{region " SIGNAL AREA : NAME->X_I_Out_ESS LENGTH->16 STARTBIT :48"}
_FB_UNPACK_WORD_TO_BYTE_6 (
		X_WORD_0										:= 
(*SELECT 1 : Is data valid and range is not exceed?*)	SEL((GVL.IOVD.X_I_Out_ESS.v AND NOT GVL.IOVD.X_I_Out_ESS.RangeExcd),
(*SELECT 2 : Is NOT AVAILABLE ?*)						SEL(GVL.IOVD.X_I_Out_ESS.na,
(*SELECT 3 : Is ERROR active ?*)						SEL(GVL.IOVD.X_I_Out_ESS.e,
(*DEFAULT VALUE assignment*)							UINT_TO_WORD(REAL_TO_UINT((32766))),
(*ERROR is active*)										16#FEFE),
(*NOT AVAILABLE is active*)								16#FFFF),
(*Transmission is VALID*)								UINT_TO_WORD(REAL_TO_UINT((GVL.IOVD.X_I_Out_ESS.x + 32766)))),
		X_BYTE_0										=> _FB_CanTx_Message_463.X_Byte_6,
		X_BYTE_1										=> _FB_CanTx_Message_463.X_Byte_7);
{endregion}

_FB_CanTx_Message_463.X_Byte_3 		:= 16#FF;

_FB_CanTx_Message_463 (		C_Enable		:= GVL.IOVD.C_En_TCU_Analog_0X463,
     						Obj_CAN			:= ADR(GVL.IC.Obj_CAN0),
     						X_MsgID			:= 16#463,
     						Tm_CycleTime	:= TIME#250MS,
     						N_Msg_Dlc		:= 8,
     						S_Extended		:= 0,
     						S_Sent_Ok   	=> GVL.IOVD.S_SentOk_TCU_Analog_0X463);
{endregion}
//-----------------------------------------------------------------------------------------------------------------------------
//-----------------------------------------------------------------------------------------------------------------------------
{region " MESSAGE AREA :TCU_Cikis_Akim_Guc- ID:464"}

{region " SIGNAL AREA : NAME->X_I_Out_Mot_Cnv LENGTH->16 STARTBIT :0"}
_FB_UNPACK_WORD_TO_BYTE_7(
		X_WORD_0										:= 
(*SELECT 1 : Is data valid and range is not exceed?*)	SEL((GVL.IOVD.X_I_Out_Mot_Cnv.v AND NOT GVL.IOVD.X_I_Out_Mot_Cnv.RangeExcd),
(*SELECT 2 : Is NOT AVAILABLE ?*)						SEL(GVL.IOVD.X_I_Out_Mot_Cnv.na,
(*SELECT 3 : Is ERROR active ?*)						SEL(GVL.IOVD.X_I_Out_Mot_Cnv.e,
(*DEFAULT VALUE assignment*)							UINT_TO_WORD(REAL_TO_UINT((1600)/0.05)),
(*ERROR is active*)										16#FEFE),
(*NOT AVAILABLE is active*)								16#FFFF),
(*Transmission is VALID*)								UINT_TO_WORD(REAL_TO_UINT((GVL.IOVD.X_I_Out_Mot_Cnv.x + 1600)/0.05))),
		X_BYTE_0										=> _FB_CanTx_Message_464.X_Byte_0,
		X_BYTE_1										=> _FB_CanTx_Message_464.X_Byte_1);
{endregion}

{region " SIGNAL AREA : NAME->X_I_Brk_Rsr LENGTH->16 STARTBIT :16"}
_FB_UNPACK_WORD_TO_BYTE_8(
		X_WORD_0										:= 
(*SELECT 1 : Is data valid and range is not exceed?*)	SEL((GVL.IOVD.X_I_Brk_Rsr.v AND NOT GVL.IOVD.X_I_Brk_Rsr.RangeExcd),
(*SELECT 2 : Is NOT AVAILABLE ?*)						SEL(GVL.IOVD.X_I_Brk_Rsr.na,
(*SELECT 3 : Is ERROR active ?*)						SEL(GVL.IOVD.X_I_Brk_Rsr.e,
(*DEFAULT VALUE assignment*)							UINT_TO_WORD(REAL_TO_UINT((1600)/0.05)),
(*ERROR is active*)										16#FEFE),
(*NOT AVAILABLE is active*)								16#FFFF),
(*Transmission is VALID*)								UINT_TO_WORD(REAL_TO_UINT((GVL.IOVD.X_I_Brk_Rsr.x + 1600)/0.05))),
		X_BYTE_0										=> _FB_CanTx_Message_464.X_Byte_2,
		X_BYTE_1										=> _FB_CanTx_Message_464.X_Byte_3);
{endregion}

{region " SIGNAL AREA : NAME->X_P_Mot_Cnv LENGTH->16 STARTBIT :32"}
_FB_UNPACK_WORD_TO_BYTE_9(
		X_WORD_0										:= 
(*SELECT 1 : Is data valid and range is not exceed?*)	SEL((GVL.IOVD.X_P_Mot_Cnv.v AND NOT GVL.IOVD.X_P_Mot_Cnv.RangeExcd),
(*SELECT 2 : Is NOT AVAILABLE ?*)						SEL(GVL.IOVD.X_P_Mot_Cnv.na,
(*SELECT 3 : Is ERROR active ?*)						SEL(GVL.IOVD.X_P_Mot_Cnv.e,
(*DEFAULT VALUE assignment*)							UINT_TO_WORD(REAL_TO_UINT((750)/0.025)),
(*ERROR is active*)										16#FEFE),
(*NOT AVAILABLE is active*)								16#FFFF),
(*Transmission is VALID*)								UINT_TO_WORD(REAL_TO_UINT((GVL.IOVD.X_P_Mot_Cnv.x + 750)/0.025))),
		X_BYTE_0										=> _FB_CanTx_Message_464.X_Byte_4,
		X_BYTE_1										=> _FB_CanTx_Message_464.X_Byte_5);
{endregion}

{region " SIGNAL AREA : NAME->X_P_Brk_Rsr LENGTH->16 STARTBIT :48"}
_FB_UNPACK_WORD_TO_BYTE_10(
		X_WORD_0										:= 
(*SELECT 1 : Is data valid and range is not exceed?*)	SEL((GVL.IOVD.X_P_Brk_Rsr.v AND NOT GVL.IOVD.X_P_Brk_Rsr.RangeExcd),
(*SELECT 2 : Is NOT AVAILABLE ?*)						SEL(GVL.IOVD.X_P_Brk_Rsr.na,
(*SELECT 3 : Is ERROR active ?*)						SEL(GVL.IOVD.X_P_Brk_Rsr.e,
(*DEFAULT VALUE assignment*)							UINT_TO_WORD(REAL_TO_UINT((750)/0.025)),
(*ERROR is active*)										16#FEFE),
(*NOT AVAILABLE is active*)								16#FFFF),
(*Transmission is VALID*)								UINT_TO_WORD(REAL_TO_UINT((GVL.IOVD.X_P_Brk_Rsr.x + 750)/0.025))),
		X_BYTE_0										=> _FB_CanTx_Message_464.X_Byte_6,
		X_BYTE_1										=> _FB_CanTx_Message_464.X_Byte_7);
{endregion}

_FB_CanTx_Message_464 (		C_Enable		:= GVL.IOVD.C_En_TCU_Cikis_Akim_Guc_0X464,
     						Obj_CAN			:= ADR(GVL.IC.Obj_CAN0),
     						X_MsgID			:= 16#464,
     						Tm_CycleTime	:= TIME#250MS,
     						N_Msg_Dlc		:= 8,
     						S_Extended		:= 0,
     						S_Sent_Ok   	=> GVL.IOVD.S_SentOk_TCU_Cikis_Akim_Guc_0X464);
{endregion}
//-----------------------------------------------------------------------------------------------------------------------------
//-----------------------------------------------------------------------------------------------------------------------------
{region " MESSAGE AREA :TCU_Tork_Hiz- ID:465"}

{region " SIGNAL AREA : NAME->X_M_Act LENGTH->16 STARTBIT :0"}
_FB_UNPACK_WORD_TO_BYTE_11 (
		X_WORD_0										:= 
(*SELECT 1 : Is data valid and range is not exceed?*)	SEL((GVL.IOVD.X_M_Act.v AND NOT GVL.IOVD.X_M_Act.RangeExcd),
(*SELECT 2 : Is NOT AVAILABLE ?*)						SEL(GVL.IOVD.X_M_Act.na,
(*SELECT 3 : Is ERROR active ?*)						SEL(GVL.IOVD.X_M_Act.e,
(*DEFAULT VALUE assignment*)							UINT_TO_WORD(REAL_TO_UINT((32766))),
(*ERROR is active*)										16#FEFE),
(*NOT AVAILABLE is active*)								16#FFFF),
(*Transmission is VALID*)								UINT_TO_WORD(REAL_TO_UINT((GVL.IOVD.X_M_Act.x + 32766)))),
		X_BYTE_0										=> _FB_CanTx_Message_465.X_Byte_0,
		X_BYTE_1										=> _FB_CanTx_Message_465.X_Byte_1);
{endregion}

{region " SIGNAL AREA : NAME->X_Spd_Act LENGTH->16 STARTBIT :16"}
_FB_UNPACK_WORD_TO_BYTE_12 (
		X_WORD_0										:= 
(*SELECT 1 : Is data valid and range is not exceed?*)	SEL((GVL.IOVD.X_Spd_Act.v AND NOT GVL.IOVD.X_Spd_Act.RangeExcd),
(*SELECT 2 : Is NOT AVAILABLE ?*)						SEL(GVL.IOVD.X_Spd_Act.na,
(*SELECT 3 : Is ERROR active ?*)						SEL(GVL.IOVD.X_Spd_Act.e,
(*DEFAULT VALUE assignment*)							UINT_TO_WORD(REAL_TO_UINT((32766))),
(*ERROR is active*)										16#FEFE),
(*NOT AVAILABLE is active*)								16#FFFF),
(*Transmission is VALID*)								UINT_TO_WORD(REAL_TO_UINT((GVL.IOVD.X_Spd_Act.x + 32766)))),
		X_BYTE_0										=> _FB_CanTx_Message_465.X_Byte_2,
		X_BYTE_1										=> _FB_CanTx_Message_465.X_Byte_3);
{endregion}

{region " SIGNAL AREA : NAME->X_Spd_Act_kmh LENGTH->16 STARTBIT :32"}
_FB_UNPACK_WORD_TO_BYTE_13 (
		X_WORD_0										:= 
(*SELECT 1 : Is data valid and range is not exceed?*)	SEL((GVL.IOVD.X_Spd_Act_kmh.v AND NOT GVL.IOVD.X_Spd_Act_kmh.RangeExcd),
(*SELECT 2 : Is NOT AVAILABLE ?*)						SEL(GVL.IOVD.X_Spd_Act_kmh.na,
(*SELECT 3 : Is ERROR active ?*)						SEL(GVL.IOVD.X_Spd_Act_kmh.e,
(*DEFAULT VALUE assignment*)							0,
(*ERROR is active*)										16#FEFE),
(*NOT AVAILABLE is active*)								16#FFFF),
(*Transmission is VALID*)								UINT_TO_WORD(REAL_TO_UINT((GVL.IOVD.X_Spd_Act_kmh.x)/0.01))),
		X_BYTE_0										=> _FB_CanTx_Message_465.X_Byte_4,
		X_BYTE_1										=> _FB_CanTx_Message_465.X_Byte_5);

{endregion}

_FB_CanTx_Message_465.X_Byte_6	:= 16#FF;
_FB_CanTx_Message_465.X_Byte_7	:= 16#FF;
	 
_FB_CanTx_Message_465 (		C_Enable		:= GVL.IOVD.C_En_TCU_Tork_Hiz_0X465,
     						Obj_CAN			:= ADR(GVL.IC.Obj_CAN0),
     						X_MsgID			:= 16#465,
     						Tm_CycleTime	:= TIME#250MS,
     						N_Msg_Dlc		:= 8,
     						S_Extended		:= 0,
     						S_Sent_Ok  	 	=> GVL.IOVD.S_SentOk_TCU_Tork_Hiz_0X465);
{endregion}
//-----------------------------------------------------------------------------------------------------------------------------
//-----------------------------------------------------------------------------------------------------------------------------
{region " MESSAGE AREA :TCU_Calisma_Suresi- ID:466"}

{region " SIGNAL AREA : NAME->N_Tm_Trol_Md LENGTH->32 STARTBIT :0"}
_FB_UNPACK_DWORD_TO_BYTE_0 (
		X_DWORD_0										:= 
(*SELECT 1 : Is data valid and range is not exceed?*)	SEL((GVL.IOVD.N_Tm_Trol_Md.v AND NOT GVL.IOVD.N_Tm_Trol_Md.RangeExcd),
(*SELECT 2 : Is NOT AVAILABLE ?*)						SEL(GVL.IOVD.N_Tm_Trol_Md.na,
(*SELECT 3 : Is ERROR active ?*)						SEL(GVL.IOVD.N_Tm_Trol_Md.e,
(*DEFAULT VALUE assignment*)							0,
(*ERROR is active*)										16#FEFEFEFE),
(*NOT AVAILABLE is active*)								16#FFFFFFFF),
(*Transmission is VALID*)								UDINT_TO_DWORD(GVL.IOVD.N_Tm_Trol_Md.x )),
		X_BYTE_0										=> _FB_CanTx_Message_466.X_Byte_0,
		X_BYTE_1										=> _FB_CanTx_Message_466.X_Byte_1,
		X_BYTE_2										=> _FB_CanTx_Message_466.X_Byte_2,
		X_BYTE_3										=> _FB_CanTx_Message_466.X_Byte_3);
{endregion}

{region " SIGNAL AREA : NAME->N_Tm_Bat_Md LENGTH->32 STARTBIT :32"}
_FB_UNPACK_DWORD_TO_BYTE_1 (
		X_DWORD_0										:= 
(*SELECT 1 : Is data valid and range is not exceed?*)	SEL((GVL.IOVD.N_Tm_Bat_Md.v AND NOT GVL.IOVD.N_Tm_Bat_Md.RangeExcd),
(*SELECT 2 : Is NOT AVAILABLE ?*)						SEL(GVL.IOVD.N_Tm_Bat_Md.na,
(*SELECT 3 : Is ERROR active ?*)						SEL(GVL.IOVD.N_Tm_Bat_Md.e,
(*DEFAULT VALUE assignment*)							0,
(*ERROR is active*)										16#FEFEFEFE),
(*NOT AVAILABLE is active*)								16#FFFFFFFF),
(*Transmission is VALID*)								UDINT_TO_DWORD(GVL.IOVD.N_Tm_Bat_Md.x )),
		X_BYTE_0										=> _FB_CanTx_Message_466.X_Byte_4,
		X_BYTE_1										=> _FB_CanTx_Message_466.X_Byte_5,
		X_BYTE_2										=> _FB_CanTx_Message_466.X_Byte_6,
		X_BYTE_3										=> _FB_CanTx_Message_466.X_Byte_7);
{endregion}

_FB_CanTx_Message_466 (		C_Enable		:= GVL.IOVD.C_En_TCU_Calisma_Suresi_0X466,
     						Obj_CAN			:= ADR(GVL.IC.Obj_CAN0),
     						X_MsgID			:= 16#466,
     						Tm_CycleTime	:= TIME#250MS,
     						N_Msg_Dlc		:= 8,
     						S_Extended		:= 0,
     						S_Sent_Ok   	=> GVL.IOVD.S_SentOk_TCU_Calisma_Suresi_0X466);
{endregion}
//-----------------------------------------------------------------------------------------------------------------------------
//-----------------------------------------------------------------------------------------------------------------------------
{region " MESSAGE AREA :TCU_Analog_2- ID:467"}

{region " SIGNAL AREA : NAME->X_U_Inv_HV LENGTH->16 STARTBIT :0"}
_FB_UNPACK_WORD_TO_BYTE_14 (
		X_WORD_0										:= 
(*SELECT 1 : Is data valid and range is not exceed?*)	SEL((GVL.IOVD.X_U_Inv_HV.v AND NOT GVL.IOVD.X_U_Inv_HV.RangeExcd),
(*SELECT 2 : Is NOT AVAILABLE ?*)						SEL(GVL.IOVD.X_U_Inv_HV.na,
(*SELECT 3 : Is ERROR active ?*)						SEL(GVL.IOVD.X_U_Inv_HV.e,
(*DEFAULT VALUE assignment*)							0,
(*ERROR is active*)										16#FEFE),
(*NOT AVAILABLE is active*)								16#FFFF),
(*Transmission is VALID*)								UINT_TO_WORD(REAL_TO_UINT((GVL.IOVD.X_U_Inv_HV.x)/0.025))),
		X_BYTE_0										=> _FB_CanTx_Message_467.X_Byte_0,
		X_BYTE_1										=> _FB_CanTx_Message_467.X_Byte_1);
{endregion}

{region " SIGNAL AREA : NAME->X_U_Cat_Ln LENGTH->16 STARTBIT :16"}
_FB_UNPACK_WORD_TO_BYTE_15 (
		X_WORD_0										:= 
(*SELECT 1 : Is data valid and range is not exceed?*)	SEL((GVL.IOVD.X_U_Cat_Ln.v AND NOT GVL.IOVD.X_U_Cat_Ln.RangeExcd),
(*SELECT 2 : Is NOT AVAILABLE ?*)						SEL(GVL.IOVD.X_U_Cat_Ln.na,
(*SELECT 3 : Is ERROR active ?*)						SEL(GVL.IOVD.X_U_Cat_Ln.e,
(*DEFAULT VALUE assignment*)							0,
(*ERROR is active*)										16#FEFE),
(*NOT AVAILABLE is active*)								16#FFFF),
(*Transmission is VALID*)								UINT_TO_WORD(REAL_TO_UINT((GVL.IOVD.X_U_Cat_Ln.x)/0.025))),
		X_BYTE_0										=> _FB_CanTx_Message_467.X_Byte_2,
		X_BYTE_1										=> _FB_CanTx_Message_467.X_Byte_3);
{endregion}

_FB_CanTx_Message_467.X_Byte_4:=16#FF;
_FB_CanTx_Message_467.X_Byte_5:=16#FF;
_FB_CanTx_Message_467.X_Byte_6:=16#FF;
_FB_CanTx_Message_467.X_Byte_7:=16#FF;
_FB_CanTx_Message_467(
     C_Enable:= GVL.IOVD.C_En_TCU_Analog_2_0X467,
     Obj_CAN:= ADR(GVL.IC.Obj_CAN0),
     X_MsgID:= 16#467,
     Tm_CycleTime:= TIME#250ms,
     N_Msg_Dlc:=8,
     S_Extended:= 0,
     S_Sent_Ok   => GVL.IOVD.S_SentOk_TCU_Analog_2_0X467);
{endregion}
//-----------------------------------------------------------------------------------------------------------------------------
//-----------------------------------------------------------------------------------------------------------------------------
{region " MESSAGE AREA :Yardimci_Konvertor_Durum- ID:480"}

{region " SIGNAL AREA : NAME->S_Aux_AC_Cnv_Rdy LENGTH->2 STARTBIT :0"}
_FB_CanTx_Message_Unpack_480.S_Bit_0		:= (GVL.IOVD.S_Aux_AC_Cnv_Rdy.x OR GVL.IOVD.S_Aux_AC_Cnv_Rdy.na) AND NOT GVL.IOVD.S_Aux_AC_Cnv_Rdy.e; 
_FB_CanTx_Message_Unpack_480.S_Bit_1		:= NOT GVL.IOVD.S_Aux_AC_Cnv_Rdy.v OR GVL.IOVD.S_Aux_AC_Cnv_Rdy.na OR GVL.IOVD.S_Aux_AC_Cnv_Rdy.e; 
{endregion}

{region " SIGNAL AREA : NAME->C_Aux_AC_Cnv_On LENGTH->2 STARTBIT :2"}
_FB_CanTx_Message_Unpack_480.S_Bit_2		:= (GVL.IOVD.C_Aux_AC_Cnv_On.x OR GVL.IOVD.C_Aux_AC_Cnv_On.na) AND NOT GVL.IOVD.C_Aux_AC_Cnv_On.e; 
_FB_CanTx_Message_Unpack_480.S_Bit_3		:= NOT GVL.IOVD.C_Aux_AC_Cnv_On.v OR GVL.IOVD.C_Aux_AC_Cnv_On.na OR GVL.IOVD.C_Aux_AC_Cnv_On.e; 
{endregion}

{region " SIGNAL AREA : NAME->S_Aux_AC_Cnv_On LENGTH->2 STARTBIT :4"}
_FB_CanTx_Message_Unpack_480.S_Bit_4		:= (GVL.IOVD.S_Aux_AC_Cnv_On.x OR GVL.IOVD.S_Aux_AC_Cnv_On.na) AND NOT GVL.IOVD.S_Aux_AC_Cnv_On.e; 
_FB_CanTx_Message_Unpack_480.S_Bit_5		:= NOT GVL.IOVD.S_Aux_AC_Cnv_On.v OR GVL.IOVD.S_Aux_AC_Cnv_On.na OR GVL.IOVD.S_Aux_AC_Cnv_On.e; 
{endregion}

{region " SIGNAL AREA : NAME->S_Aux_DC_24V_Cnv_Rdy LENGTH->2 STARTBIT :6"}
_FB_CanTx_Message_Unpack_480.S_Bit_6		:= (GVL.IOVD.S_Aux_DC_24V_Cnv_Rdy.x OR GVL.IOVD.S_Aux_DC_24V_Cnv_Rdy.na) AND NOT GVL.IOVD.S_Aux_DC_24V_Cnv_Rdy.e; 
_FB_CanTx_Message_Unpack_480.S_Bit_7		:= NOT GVL.IOVD.S_Aux_DC_24V_Cnv_Rdy.v OR GVL.IOVD.S_Aux_DC_24V_Cnv_Rdy.na OR GVL.IOVD.S_Aux_DC_24V_Cnv_Rdy.e; 
{endregion}

{region " SIGNAL AREA : NAME->C_Aux_DC_24V_Cnv_On LENGTH->2 STARTBIT :8"}
_FB_CanTx_Message_Unpack_480.S_Bit_8		:= (GVL.IOVD.C_Aux_DC_24V_Cnv_On.x OR GVL.IOVD.C_Aux_DC_24V_Cnv_On.na) AND NOT GVL.IOVD.C_Aux_DC_24V_Cnv_On.e; 
_FB_CanTx_Message_Unpack_480.S_Bit_9		:=  NOT GVL.IOVD.C_Aux_DC_24V_Cnv_On.v OR GVL.IOVD.C_Aux_DC_24V_Cnv_On.na OR GVL.IOVD.C_Aux_DC_24V_Cnv_On.e; 
{endregion}

{region " SIGNAL AREA : NAME->S_Aux_DC_24V_Cnv_On LENGTH->2 STARTBIT :10"}
_FB_CanTx_Message_Unpack_480.S_Bit_10		:= (GVL.IOVD.S_Aux_DC_24V_Cnv_On.x OR GVL.IOVD.S_Aux_DC_24V_Cnv_On.na) AND NOT GVL.IOVD.S_Aux_DC_24V_Cnv_On.e; 
_FB_CanTx_Message_Unpack_480.S_Bit_11		:= NOT GVL.IOVD.S_Aux_DC_24V_Cnv_On.v OR GVL.IOVD.S_Aux_DC_24V_Cnv_On.na OR GVL.IOVD.S_Aux_DC_24V_Cnv_On.e; 
{endregion}

{region " SIGNAL AREA : NAME->C_Aux_DC_Cnv_On LENGTH->2 STARTBIT :12"}
_FB_CanTx_Message_Unpack_480.S_Bit_12		:= (GVL.IOVD.C_Aux_DC_Cnv_On.x OR GVL.IOVD.C_Aux_DC_Cnv_On.na) AND NOT GVL.IOVD.C_Aux_DC_Cnv_On.e; 
_FB_CanTx_Message_Unpack_480.S_Bit_13		:= NOT GVL.IOVD.C_Aux_DC_Cnv_On.v OR GVL.IOVD.C_Aux_DC_Cnv_On.na OR GVL.IOVD.C_Aux_DC_Cnv_On.e; 
{endregion}

{region " SIGNAL AREA : NAME->S_Aux_DC_Cnv_On LENGTH->2 STARTBIT :14"}
_FB_CanTx_Message_Unpack_480.S_Bit_14		:= (GVL.IOVD.S_Aux_DC_Cnv_On.x OR GVL.IOVD.S_Aux_DC_Cnv_On.na) AND NOT GVL.IOVD.S_Aux_DC_Cnv_On.e; 
_FB_CanTx_Message_Unpack_480.S_Bit_15		:= NOT GVL.IOVD.S_Aux_DC_Cnv_On.v OR GVL.IOVD.S_Aux_DC_Cnv_On.na OR GVL.IOVD.S_Aux_DC_Cnv_On.e; 
{endregion}

{region " SIGNAL AREA : NAME->C_Bat_Chrg_DC_Cnv_On LENGTH->2 STARTBIT :16"}
_FB_CanTx_Message_Unpack_480.S_Bit_16		:= (GVL.IOVD.C_Bat_Chrg_DC_Cnv_On.x OR GVL.IOVD.C_Bat_Chrg_DC_Cnv_On.na) AND NOT GVL.IOVD.C_Bat_Chrg_DC_Cnv_On.e; 
_FB_CanTx_Message_Unpack_480.S_Bit_17		:= NOT GVL.IOVD.C_Bat_Chrg_DC_Cnv_On.v OR GVL.IOVD.C_Bat_Chrg_DC_Cnv_On.na OR GVL.IOVD.C_Bat_Chrg_DC_Cnv_On.e; 
{endregion}

{region " SIGNAL AREA : NAME->S_Bat_Chrg_DC_Cnv_On LENGTH->2 STARTBIT :18"}
_FB_CanTx_Message_Unpack_480.S_Bit_18		:= (GVL.IOVD.S_Bat_Chrg_DC_Cnv_On.x OR GVL.IOVD.S_Bat_Chrg_DC_Cnv_On.na) AND NOT GVL.IOVD.S_Bat_Chrg_DC_Cnv_On.e; 
_FB_CanTx_Message_Unpack_480.S_Bit_19		:= NOT GVL.IOVD.S_Bat_Chrg_DC_Cnv_On.v OR GVL.IOVD.S_Bat_Chrg_DC_Cnv_On.na OR GVL.IOVD.S_Bat_Chrg_DC_Cnv_On.e; 
{endregion}

{region " SIGNAL AREA : NAME->C_Aux_DC_Ct_1_On LENGTH->2 STARTBIT :20"}
_FB_CanTx_Message_Unpack_480.S_Bit_20		:= (GVL.IOVD.C_Aux_DC_Ct_1_On.x OR GVL.IOVD.C_Aux_DC_Ct_1_On.na) AND NOT GVL.IOVD.C_Aux_DC_Ct_1_On.e; 
_FB_CanTx_Message_Unpack_480.S_Bit_21		:= NOT GVL.IOVD.C_Aux_DC_Ct_1_On.v OR GVL.IOVD.C_Aux_DC_Ct_1_On.na OR GVL.IOVD.C_Aux_DC_Ct_1_On.e; 
{endregion}

{region " SIGNAL AREA : NAME->C_Aux_DC_Ct_2_On LENGTH->2 STARTBIT :22"}
_FB_CanTx_Message_Unpack_480.S_Bit_22		:= (GVL.IOVD.C_Aux_DC_Ct_2_On.x OR GVL.IOVD.C_Aux_DC_Ct_2_On.na) AND NOT GVL.IOVD.C_Aux_DC_Ct_2_On.e; 
_FB_CanTx_Message_Unpack_480.S_Bit_23		:= NOT GVL.IOVD.C_Aux_DC_Ct_2_On.v OR GVL.IOVD.C_Aux_DC_Ct_2_On.na OR GVL.IOVD.C_Aux_DC_Ct_2_On.e; 
{endregion}

{region " SIGNAL AREA : NAME->C_Aux_DC_Ct_3_On LENGTH->2 STARTBIT :24"}
_FB_CanTx_Message_Unpack_480.S_Bit_24		:= (GVL.IOVD.C_Aux_DC_Ct_3_On.x OR GVL.IOVD.C_Aux_DC_Ct_3_On.na) AND NOT GVL.IOVD.C_Aux_DC_Ct_3_On.e; 
_FB_CanTx_Message_Unpack_480.S_Bit_25		:= NOT GVL.IOVD.C_Aux_DC_Ct_3_On.v OR GVL.IOVD.C_Aux_DC_Ct_3_On.na OR GVL.IOVD.C_Aux_DC_Ct_3_On.e; 
{endregion}

{region " SIGNAL AREA : NAME->S_Aux_DC_Ct_1_Actv LENGTH->2 STARTBIT :26"}
_FB_CanTx_Message_Unpack_480.S_Bit_26		:= (GVL.IOVD.S_Aux_DC_Ct_1_Actv.x OR GVL.IOVD.S_Aux_DC_Ct_1_Actv.na) AND NOT GVL.IOVD.S_Aux_DC_Ct_1_Actv.e; 
_FB_CanTx_Message_Unpack_480.S_Bit_27		:= NOT GVL.IOVD.S_Aux_DC_Ct_1_Actv.v OR GVL.IOVD.S_Aux_DC_Ct_1_Actv.na OR GVL.IOVD.S_Aux_DC_Ct_1_Actv.e; 
{endregion}

{region " SIGNAL AREA : NAME->S_Aux_DC_Ct_2_Actv LENGTH->2 STARTBIT :28"}
_FB_CanTx_Message_Unpack_480.S_Bit_28		:= (GVL.IOVD.S_Aux_DC_Ct_2_Actv.x OR GVL.IOVD.S_Aux_DC_Ct_2_Actv.na) AND NOT GVL.IOVD.S_Aux_DC_Ct_2_Actv.e; 
_FB_CanTx_Message_Unpack_480.S_Bit_29		:=	NOT GVL.IOVD.S_Aux_DC_Ct_2_Actv.v OR GVL.IOVD.S_Aux_DC_Ct_2_Actv.na OR GVL.IOVD.S_Aux_DC_Ct_2_Actv.e; 
{endregion}

{region " SIGNAL AREA : NAME->S_Aux_DC_Ct_3_Actv LENGTH->2 STARTBIT :30"}
_FB_CanTx_Message_Unpack_480.S_Bit_30		:= (GVL.IOVD.S_Aux_DC_Ct_3_Actv.x OR GVL.IOVD.S_Aux_DC_Ct_3_Actv.na) AND NOT GVL.IOVD.S_Aux_DC_Ct_3_Actv.e; 
_FB_CanTx_Message_Unpack_480.S_Bit_31		:= NOT GVL.IOVD.S_Aux_DC_Ct_3_Actv.v OR GVL.IOVD.S_Aux_DC_Ct_3_Actv.na OR GVL.IOVD.S_Aux_DC_Ct_3_Actv.e; 
{endregion}

{region " SIGNAL AREA : NAME->Z_Bccu_Stat LENGTH->8 STARTBIT :32"}
_FB_CanTx_Message_Unpack_480.X_Byte_4					:=
(*SELECT 1 : Is data valid and range is not exceed?*)	SEL((GVL.IOVD.Z_Bccu_Stat.v AND NOT GVL.IOVD.Z_Bccu_Stat.RangeExcd),
(*SELECT 2 : Is NOT AVAILABLE ?*)						SEL(GVL.IOVD.Z_Bccu_Stat.na,
(*SELECT 3 : Is ERROR active ?*)						SEL(GVL.IOVD.Z_Bccu_Stat.e,
(*DEFAULT VALUE assignment*)							0,
(*ERROR is active*)										16#FE),
(*NOT AVAILABLE is active*)								16#FF),
(*Transmission is VALID*)								GVL.IOVD.Z_Bccu_Stat.x);
{endregion}

{region " SIGNAL AREA : NAME->Z_Tcu_Stat LENGTH->8 STARTBIT :32"}
_FB_CanTx_Message_Unpack_480.X_Byte_5					:=
(*SELECT 1 : Is data valid and range is not exceed?*)	SEL((GVL.IOVD.Z_Tcu_Stat.v AND NOT GVL.IOVD.Z_Tcu_Stat.RangeExcd),
(*SELECT 2 : Is NOT AVAILABLE ?*)						SEL(GVL.IOVD.Z_Tcu_Stat.na,
(*SELECT 3 : Is ERROR active ?*)						SEL(GVL.IOVD.Z_Tcu_Stat.e,
(*DEFAULT VALUE assignment*)							0,
(*ERROR is active*)										16#FE),
(*NOT AVAILABLE is active*)								16#FF),
(*Transmission is VALID*)								GVL.IOVD.Z_Tcu_Stat.x);
{endregion}	

{region " SIGNAL AREA : NAME->Z_Apu_Stat LENGTH->8 STARTBIT :32"}
_FB_CanTx_Message_Unpack_480.X_Byte_6					:=
(*SELECT 1 : Is data valid and range is not exceed?*)	SEL((GVL.IOVD.Z_Apu_Stat.v AND NOT GVL.IOVD.Z_Apu_Stat.RangeExcd),
(*SELECT 2 : Is NOT AVAILABLE ?*)						SEL(GVL.IOVD.Z_Apu_Stat.na,
(*SELECT 3 : Is ERROR active ?*)						SEL(GVL.IOVD.Z_Apu_Stat.e,
(*DEFAULT VALUE assignment*)							0,
(*ERROR is active*)										16#FE),
(*NOT AVAILABLE is active*)								16#FF),
(*Transmission is VALID*)								GVL.IOVD.Z_Apu_Stat.x);
{endregion}			   

_FB_CanTx_Message_Unpack_480.X_Byte_7	:= 16#FF;

_FB_CanTx_Message_Unpack_480 (		C_Enable		:= GVL.IOVD.C_En_Yardimci_Konvertor_Durum_0X480,
     								Obj_CAN			:= ADR(GVL.IC.Obj_CAN0),
     								X_MsgID			:= 16#480,
     								Tm_CycleTime	:= TIME#250MS,
     								N_Msg_Dlc		:= 8,
     								S_Extended		:= 0,
     								S_Sent_Ok   	=> GVL.IOVD.S_SentOk_Yardimci_Konvertor_Durum_0X480);
{endregion}
//-----------------------------------------------------------------------------------------------------------------------------
//-----------------------------------------------------------------------------------------------------------------------------
{region " MESSAGE AREA :Yardimci_Konvertor_Akim- ID:481"}

{region " SIGNAL AREA : NAME->X_I_Out_Aux_DC_Cnv LENGTH->16 STARTBIT :0"}
_FB_UNPACK_WORD_TO_BYTE_16 (
		X_WORD_0										:= 
(*SELECT 1 : Is data valid and range is not exceed?*)	SEL((GVL.IOVD.X_I_Out_Aux_DC_Cnv.v AND NOT GVL.IOVD.X_I_Out_Aux_DC_Cnv.RangeExcd),
(*SELECT 2 : Is NOT AVAILABLE ?*)						SEL(GVL.IOVD.X_I_Out_Aux_DC_Cnv.na,
(*SELECT 3 : Is ERROR active ?*)						SEL(GVL.IOVD.X_I_Out_Aux_DC_Cnv.e,
(*DEFAULT VALUE assignment*)							0,
(*ERROR is active*)										16#FEFE),
(*NOT AVAILABLE is active*)								16#FFFF),
(*Transmission is VALID*)								UINT_TO_WORD(REAL_TO_UINT((GVL.IOVD.X_I_Out_Aux_DC_Cnv.x)/0.1))),
		X_BYTE_0										=> _FB_CanTx_Message_Unpack_481.X_Byte_0,
		X_BYTE_1										=> _FB_CanTx_Message_Unpack_481.X_Byte_1);
{endregion}

{region " SIGNAL AREA : NAME->X_I_Out_Aux_AC_Cnv LENGTH->16 STARTBIT :16"}
_FB_UNPACK_WORD_TO_BYTE_17 (
		X_WORD_0										:= 
(*SELECT 1 : Is data valid and range is not exceed?*)	SEL((GVL.IOVD.X_I_Out_Aux_AC_Cnv.v AND NOT GVL.IOVD.X_I_Out_Aux_AC_Cnv.RangeExcd),
(*SELECT 2 : Is NOT AVAILABLE ?*)						SEL(GVL.IOVD.X_I_Out_Aux_AC_Cnv.na,
(*SELECT 3 : Is ERROR active ?*)						SEL(GVL.IOVD.X_I_Out_Aux_AC_Cnv.e,
(*DEFAULT VALUE assignment*)							0,
(*ERROR is active*)										16#FEFE),
(*NOT AVAILABLE is active*)								16#FFFF),
(*Transmission is VALID*)								UINT_TO_WORD(REAL_TO_UINT((GVL.IOVD.X_I_Out_Aux_AC_Cnv.x)/0.1))),
		X_BYTE_0										=> _FB_CanTx_Message_Unpack_481.X_Byte_2,
		X_BYTE_1										=> _FB_CanTx_Message_Unpack_481.X_Byte_3);
{endregion}

{region " SIGNAL AREA : NAME->X_I_Out_Aux_DC_24V_Cnv LENGTH->16 STARTBIT :32"}
_FB_UNPACK_WORD_TO_BYTE_18 (
		X_WORD_0										:= 
(*SELECT 1 : Is data valid and range is not exceed?*)	SEL((GVL.IOVD.X_I_Out_Aux_DC_24V_Cnv.v AND NOT GVL.IOVD.X_I_Out_Aux_DC_24V_Cnv.RangeExcd),
(*SELECT 2 : Is NOT AVAILABLE ?*)						SEL(GVL.IOVD.X_I_Out_Aux_DC_24V_Cnv.na,
(*SELECT 3 : Is ERROR active ?*)						SEL(GVL.IOVD.X_I_Out_Aux_DC_24V_Cnv.e,
(*DEFAULT VALUE assignment*)							UINT_TO_WORD(REAL_TO_UINT((750)/0.025)),
(*ERROR is active*)										16#FEFE),
(*NOT AVAILABLE is active*)								16#FFFF),
(*Transmission is VALID*)								UINT_TO_WORD(REAL_TO_UINT((GVL.IOVD.X_I_Out_Aux_DC_24V_Cnv.x + 750)/0.025))),
		X_BYTE_0										=> _FB_CanTx_Message_Unpack_481.X_Byte_4,
		X_BYTE_1										=> _FB_CanTx_Message_Unpack_481.X_Byte_5);
{endregion}

{region " SIGNAL AREA : NAME->X_I_In_Aux_DC_24V_Cnv LENGTH->16 STARTBIT :48"}
_FB_UNPACK_WORD_TO_BYTE_19 (
		X_WORD_0										:= 
(*SELECT 1 : Is data valid and range is not exceed?*)	SEL((GVL.IOVD.X_I_In_Aux_DC_24V_Cnv.v AND NOT GVL.IOVD.X_I_In_Aux_DC_24V_Cnv.RangeExcd),
(*SELECT 2 : Is NOT AVAILABLE ?*)						SEL(GVL.IOVD.X_I_In_Aux_DC_24V_Cnv.na,
(*SELECT 3 : Is ERROR active ?*)						SEL(GVL.IOVD.X_I_In_Aux_DC_24V_Cnv.e,
(*DEFAULT VALUE assignment*)							0,
(*ERROR is active*)										16#FEFE),
(*NOT AVAILABLE is active*)								16#FFFF),
(*Transmission is VALID*)								UINT_TO_WORD(REAL_TO_UINT((GVL.IOVD.X_I_In_Aux_DC_24V_Cnv.x)/0.1))),
		X_BYTE_0										=> _FB_CanTx_Message_Unpack_481.X_Byte_6,
		X_BYTE_1										=> _FB_CanTx_Message_Unpack_481.X_Byte_7);
{endregion}

_FB_CanTx_Message_Unpack_481(
     C_Enable:= GVL.IOVD.C_En_Yardimci_Konvertor_Akim_0X481,
     Obj_CAN:= ADR(GVL.IC.Obj_CAN0),
     X_MsgID:= 16#481,
     Tm_CycleTime:= TIME#250ms,
     N_Msg_Dlc:=8,
     S_Extended:= 0,
     S_Sent_Ok   => GVL.IOVD.S_SentOk_Yardimci_Konvertor_Akim_0X481);
{endregion}
//-----------------------------------------------------------------------------------------------------------------------------
//-----------------------------------------------------------------------------------------------------------------------------
{region " MESSAGE AREA :Yardimci_Konvertor_Guc- ID:482"}

{region " SIGNAL AREA : NAME->X_U_Out_24V_Bat LENGTH->16 STARTBIT :0"}
_FB_UNPACK_WORD_TO_BYTE_20 (
		X_WORD_0										:= 
(*SELECT 1 : Is data valid and range is not exceed?*)	SEL((GVL.IOVD.X_U_Out_24V_Bat.v AND NOT GVL.IOVD.X_U_Out_24V_Bat.RangeExcd),
(*SELECT 2 : Is NOT AVAILABLE ?*)						SEL(GVL.IOVD.X_U_Out_24V_Bat.na,
(*SELECT 3 : Is ERROR active ?*)						SEL(GVL.IOVD.X_U_Out_24V_Bat.e,
(*DEFAULT VALUE assignment*)							0,
(*ERROR is active*)										16#FEFE),
(*NOT AVAILABLE is active*)								16#FFFF),
(*Transmission is VALID*)								UINT_TO_WORD(REAL_TO_UINT((GVL.IOVD.X_U_Out_24V_Bat.x)/0.01))),
		X_BYTE_0										=> _FB_CanTx_Message_Unpack_482.X_Byte_0,
		X_BYTE_1										=> _FB_CanTx_Message_Unpack_482.X_Byte_1);
{endregion}

{region " SIGNAL AREA : NAME->X_P_Out_Aux_DC_Cnv LENGTH->16 STARTBIT :16"}
_FB_UNPACK_WORD_TO_BYTE_21 (
		X_WORD_0										:= 
(*SELECT 1 : Is data valid and range is not exceed?*)	SEL((GVL.IOVD.X_P_Out_Aux_DC_Cnv.v AND NOT GVL.IOVD.X_P_Out_Aux_DC_Cnv.RangeExcd),
(*SELECT 2 : Is NOT AVAILABLE ?*)						SEL(GVL.IOVD.X_P_Out_Aux_DC_Cnv.na,
(*SELECT 3 : Is ERROR active ?*)						SEL(GVL.IOVD.X_P_Out_Aux_DC_Cnv.e,
(*DEFAULT VALUE assignment*)							UINT_TO_WORD(REAL_TO_UINT((750)/0.025)),
(*ERROR is active*)										16#FEFE),
(*NOT AVAILABLE is active*)								16#FFFF),
(*Transmission is VALID*)								UINT_TO_WORD(REAL_TO_UINT((GVL.IOVD.X_P_Out_Aux_DC_Cnv.x + 750)/0.025))),
		X_BYTE_0										=> _FB_CanTx_Message_Unpack_482.X_Byte_2,
		X_BYTE_1										=> _FB_CanTx_Message_Unpack_482.X_Byte_3);
{endregion}

{region " SIGNAL AREA : NAME->X_P_Out_Aux_AC_Cnv LENGTH->16 STARTBIT :32"}
_FB_UNPACK_WORD_TO_BYTE_22 (
		X_WORD_0										:= 
(*SELECT 1 : Is data valid and range is not exceed?*)	SEL((GVL.IOVD.X_P_Out_Aux_AC_Cnv.v AND NOT GVL.IOVD.X_P_Out_Aux_AC_Cnv.RangeExcd),
(*SELECT 2 : Is NOT AVAILABLE ?*)						SEL(GVL.IOVD.X_P_Out_Aux_AC_Cnv.na,
(*SELECT 3 : Is ERROR active ?*)						SEL(GVL.IOVD.X_P_Out_Aux_AC_Cnv.e,
(*DEFAULT VALUE assignment*)							UINT_TO_WORD(REAL_TO_UINT((750)/0.025)),
(*ERROR is active*)										16#FEFE),
(*NOT AVAILABLE is active*)								16#FFFF),
(*Transmission is VALID*)								UINT_TO_WORD(REAL_TO_UINT((GVL.IOVD.X_P_Out_Aux_AC_Cnv.x + 750)/0.025))),
		X_BYTE_0										=> _FB_CanTx_Message_Unpack_482.X_Byte_4,
		X_BYTE_1										=> _FB_CanTx_Message_Unpack_482.X_Byte_5);

{endregion}

{region " SIGNAL AREA : NAME->X_P_Out_Aux_DC_24V_Cnv LENGTH->16 STARTBIT :48"}
_FB_UNPACK_WORD_TO_BYTE_23 (
		X_WORD_0										:= 
(*SELECT 1 : Is data valid and range is not exceed?*)	SEL((GVL.IOVD.X_P_Out_Aux_DC_24V_Cnv.v AND NOT GVL.IOVD.X_P_Out_Aux_DC_24V_Cnv.RangeExcd),
(*SELECT 2 : Is NOT AVAILABLE ?*)						SEL(GVL.IOVD.X_P_Out_Aux_DC_24V_Cnv.na,
(*SELECT 3 : Is ERROR active ?*)						SEL(GVL.IOVD.X_P_Out_Aux_DC_24V_Cnv.e,
(*DEFAULT VALUE assignment*)							UINT_TO_WORD(REAL_TO_UINT((750)/0.025)),
(*ERROR is active*)										16#FEFE),
(*NOT AVAILABLE is active*)								16#FFFF),
(*Transmission is VALID*)								UINT_TO_WORD(REAL_TO_UINT((GVL.IOVD.X_P_Out_Aux_DC_24V_Cnv.x + 750)/0.025))),
		X_BYTE_0										=> _FB_CanTx_Message_Unpack_482.X_Byte_6,
		X_BYTE_1										=> _FB_CanTx_Message_Unpack_482.X_Byte_7);
{endregion}

_FB_CanTx_Message_Unpack_482 (		C_Enable		:= GVL.IOVD.C_En_Yardimci_Konvertor_Guc_0X482,
     								Obj_CAN			:= ADR(GVL.IC.Obj_CAN0),
     								X_MsgID			:= 16#482,
     								Tm_CycleTime	:= TIME#250MS,
     								N_Msg_Dlc		:= 8,
     								S_Extended		:= 0,
     								S_Sent_Ok   	=> GVL.IOVD.S_SentOk_Yardimci_Konvertor_Guc_0X482);
{endregion}
//-----------------------------------------------------------------------------------------------------------------------------
//-----------------------------------------------------------------------------------------------------------------------------
{region " MESSAGE AREA :Batarya_Sarj_Konvertor- ID:483"}

{region " SIGNAL AREA : NAME->X_P_Bat_Chrg_DC_Cnv LENGTH->16 STARTBIT :0"}
_FB_UNPACK_WORD_TO_BYTE_26 (
		X_WORD_0										:= 
(*SELECT 1 : Is data valid and range is not exceed?*)	SEL((GVL.IOVD.X_P_Bat_Chrg_DC_Cnv.v AND NOT GVL.IOVD.X_P_Bat_Chrg_DC_Cnv.RangeExcd),
(*SELECT 2 : Is NOT AVAILABLE ?*)						SEL(GVL.IOVD.X_P_Bat_Chrg_DC_Cnv.na,
(*SELECT 3 : Is ERROR active ?*)						SEL(GVL.IOVD.X_P_Bat_Chrg_DC_Cnv.e,
(*DEFAULT VALUE assignment*)							0,
(*ERROR is active*)										16#FEFE),
(*NOT AVAILABLE is active*)								16#FFFF),
(*Transmission is VALID*)								UINT_TO_WORD(REAL_TO_UINT((GVL.IOVD.X_P_Bat_Chrg_DC_Cnv.x + 3276.6)/0.1))),
		X_BYTE_0										=> _FB_CanTx_Message_Unpack_483.X_Byte_0,
		X_BYTE_1										=> _FB_CanTx_Message_Unpack_483.X_Byte_1);
{endregion}

{region " SIGNAL AREA : NAME->X_I_Out_Aux_Bat_Chrg_DC_Cnv LENGTH->16 STARTBIT :16"}
_FB_UNPACK_WORD_TO_BYTE_27 (
		X_WORD_0										:= 
(*SELECT 1 : Is data valid and range is not exceed?*)	SEL((GVL.IOVD.X_I_Out_Aux_Bat_Chrg_DC_Cnv.v AND NOT GVL.IOVD.X_I_Out_Aux_Bat_Chrg_DC_Cnv.RangeExcd),
(*SELECT 2 : Is NOT AVAILABLE ?*)						SEL(GVL.IOVD.X_I_Out_Aux_Bat_Chrg_DC_Cnv.na,
(*SELECT 3 : Is ERROR active ?*)						SEL(GVL.IOVD.X_I_Out_Aux_Bat_Chrg_DC_Cnv.e,
(*DEFAULT VALUE assignment*)							UINT_TO_WORD(REAL_TO_UINT((1600)/0.05)),
(*ERROR is active*)										16#FEFE),
(*NOT AVAILABLE is active*)								16#FFFF),
(*Transmission is VALID*)								UINT_TO_WORD(REAL_TO_UINT((GVL.IOVD.X_I_Out_Aux_Bat_Chrg_DC_Cnv.x + 1600)/0.05))),
		X_BYTE_0										=> _FB_CanTx_Message_Unpack_483.X_Byte_2,
		X_BYTE_1										=> _FB_CanTx_Message_Unpack_483.X_Byte_3);
{endregion}

_FB_CanTx_Message_Unpack_483.X_Byte_4		:= 16#FF;
_FB_CanTx_Message_Unpack_483.X_Byte_5		:= 16#FF;
_FB_CanTx_Message_Unpack_483.X_Byte_6		:= 16#FF;
_FB_CanTx_Message_Unpack_483.X_Byte_7		:= 16#FF; 

_FB_CanTx_Message_Unpack_483 (		C_Enable		:= GVL.IOVD.C_En_Batarya_Sarj_Konvertor_Analog_0X483,
     								Obj_CAN			:= ADR(GVL.IC.Obj_CAN0),
     								X_MsgID			:= 16#483,
     								Tm_CycleTime	:= TIME#250MS,
     								N_Msg_Dlc		:= 8,
     								S_Extended		:= 0,
     								S_Sent_Ok   	=> GVL.IOVD.S_SentOk_Batarya_Konvertor_Analog_0X483);
{endregion}

{region " MESSAGE AREA :Yardimci_Konvertor_Sicaklik- ID:484"}

{region " SIGNAL AREA : NAME->X_T_Aux_AC_Cnv LENGTH->8 STARTBIT :0"}
_FB_CanTx_Message_Unpack_484.X_Byte_0					:=
(*SELECT 1 : Is data valid and range is not exceed?*)	SEL((GVL.IOVD.X_T_Aux_AC_Cnv.v AND NOT GVL.IOVD.X_T_Aux_AC_Cnv.RangeExcd),
(*SELECT 2 : Is NOT AVAILABLE ?*)						SEL(GVL.IOVD.X_T_Aux_AC_Cnv.na,
(*SELECT 3 : Is ERROR active ?*)						SEL(GVL.IOVD.X_T_Aux_AC_Cnv.e,
(*DEFAULT VALUE assignment*)							USINT_TO_BYTE(REAL_TO_USINT((40))),
(*ERROR is active*)										16#FE),
(*NOT AVAILABLE is active*)								16#FF),
(*Transmission is VALID*)								USINT_TO_BYTE(REAL_TO_USINT((GVL.IOVD.X_T_Aux_AC_Cnv.x + 40))));
{endregion}

{region " SIGNAL AREA : NAME->X_T_Aux_DC_24V_Cnv LENGTH->8 STARTBIT :8"}
_FB_CanTx_Message_Unpack_484.X_Byte_1					:=
(*SELECT 1 : Is data valid and range is not exceed?*)	SEL((GVL.IOVD.X_T_Aux_DC_24V_Cnv.v AND NOT GVL.IOVD.X_T_Aux_DC_24V_Cnv.RangeExcd),
(*SELECT 2 : Is NOT AVAILABLE ?*)						SEL(GVL.IOVD.X_T_Aux_DC_24V_Cnv.na,
(*SELECT 3 : Is ERROR active ?*)						SEL(GVL.IOVD.X_T_Aux_DC_24V_Cnv.e,
(*DEFAULT VALUE assignment*)							USINT_TO_BYTE(REAL_TO_USINT((40))),
(*ERROR is active*)										16#FE),
(*NOT AVAILABLE is active*)								16#FF),
(*Transmission is VALID*)								USINT_TO_BYTE(REAL_TO_USINT((GVL.IOVD.X_T_Aux_DC_24V_Cnv.x + 40))));
{endregion}

{region " SIGNAL AREA : NAME->X_T_Aux_DC_Cnv LENGTH->8 STARTBIT :16"}
_FB_CanTx_Message_Unpack_484.X_Byte_2					:=
(*SELECT 1 : Is data valid and range is not exceed?*)	SEL((GVL.IOVD.X_T_Aux_DC_Cnv.v AND NOT GVL.IOVD.X_T_Aux_DC_Cnv.RangeExcd),
(*SELECT 2 : Is NOT AVAILABLE ?*)						SEL(GVL.IOVD.X_T_Aux_DC_Cnv.na,
(*SELECT 3 : Is ERROR active ?*)						SEL(GVL.IOVD.X_T_Aux_DC_Cnv.e,
(*DEFAULT VALUE assignment*)							USINT_TO_BYTE(REAL_TO_USINT((40))),
(*ERROR is active*)										16#FE),
(*NOT AVAILABLE is active*)								16#FF),
(*Transmission is VALID*)								USINT_TO_BYTE(REAL_TO_USINT((GVL.IOVD.X_T_Aux_DC_Cnv.x + 40))));
{endregion}

{region " SIGNAL AREA : NAME->X_T_Bat_Chrg_DC_Cnv LENGTH->8 STARTBIT :24"}
_FB_CanTx_Message_Unpack_484.X_Byte_3					:=
(*SELECT 1 : Is data valid and range is not exceed?*)	SEL((GVL.IOVD.X_T_Bat_Chrg_DC_Cnv.v AND NOT GVL.IOVD.X_T_Bat_Chrg_DC_Cnv.RangeExcd),
(*SELECT 2 : Is NOT AVAILABLE ?*)						SEL(GVL.IOVD.X_T_Bat_Chrg_DC_Cnv.na,
(*SELECT 3 : Is ERROR active ?*)						SEL(GVL.IOVD.X_T_Bat_Chrg_DC_Cnv.e,
(*DEFAULT VALUE assignment*)							USINT_TO_BYTE(REAL_TO_USINT((40))),
(*ERROR is active*)										16#FE),
(*NOT AVAILABLE is active*)								16#FF),
(*Transmission is VALID*)								USINT_TO_BYTE(REAL_TO_USINT((GVL.IOVD.X_T_Bat_Chrg_DC_Cnv.x + 40))));
{endregion}

_FB_CanTx_Message_Unpack_484.X_Byte_4	:= 16#FF;
_FB_CanTx_Message_Unpack_484.X_Byte_5	:= 16#FF;
_FB_CanTx_Message_Unpack_484.X_Byte_6	:= 16#FF;
_FB_CanTx_Message_Unpack_484.X_Byte_7	:= 16#FF;
	 
_FB_CanTx_Message_Unpack_484 (		C_Enable		:= GVL.IOVD.C_En_Yardimci_Konvertor_Sicaklik_0X484,
     								Obj_CAN			:= ADR(GVL.IC.Obj_CAN0),
     								X_MsgID			:= 16#484,
     								Tm_CycleTime	:= TIME#250MS,
     								N_Msg_Dlc		:= 8,
     								S_Extended		:= 0,
     								S_Sent_Ok   	=> GVL.IOVD.S_SentOk_Yardimci_Konvertor_Sicaklik_0X484);
{endregion}
//-----------------------------------------------------------------------------------------------------------------------------
//-----------------------------------------------------------------------------------------------------------------------------

{region " MESSAGE AREA :Isolation_Status - ID:485"}

{region " SIGNAL AREA : NAME->Z_Insu_Dev LENGTH->4 STARTBIT :0"}
_FB_UNPACK_BYTE_TO_8BITS_2(
		S_Bit_0=> _FB_CanTx_Message_Unpack_485.S_Bit_0,
		S_Bit_1=> _FB_CanTx_Message_Unpack_485.S_Bit_1,
		S_Bit_2=> _FB_CanTx_Message_Unpack_485.S_Bit_2,
		S_Bit_3=> _FB_CanTx_Message_Unpack_485.S_Bit_3,
		X_BYTE_0:=
(*SELECT 1 : Is data valid and range is not exceed?*)	SEL((GVL.IOVD.Z_Insu_Dev.v AND NOT GVL.IOVD.Z_Insu_Dev.RangeExcd),
(*SELECT 2 : Is NOT AVAILABLE ?*)						SEL(GVL.IOVD.Z_Insu_Dev.na,
(*SELECT 3 : Is ERROR active ?*)						SEL(GVL.IOVD.Z_Insu_Dev.e,
(*DEFAULT VALUE assignment*)							0,
(*ERROR is active*)										16#E),
(*NOT AVAILABLE is active*)								16#F),
(*Transmission is VALID*)								GVL.IOVD.Z_Insu_Dev.x));
{endregion}

{region " SIGNAL AREA : NAME->S_ER_Insu_Dev_Not_Conn LENGTH->1 STARTBIT :4"}
_FB_CanTx_Message_Unpack_485.S_Bit_4		:= GVL.IOVD.S_ER_Insu_Dev_Not_Conn.x AND GVL.IOVD.S_ER_Insu_Dev_Not_Conn.v;
{endregion}

{region " SIGNAL AREA : NAME->Z_Man_Insu_Tst LENGTH->8 STARTBIT :8"}
_FB_CanTx_Message_Unpack_485.X_Byte_1:=					SEL((GVL.IOVD.Z_Man_Insu_Tst.v AND NOT GVL.IOVD.Z_Man_Insu_Tst.RangeExcd),
(*SELECT 2 : Is NOT AVAILABLE ?*)						SEL(GVL.IOVD.Z_Man_Insu_Tst.na,
(*SELECT 3 : Is ERROR active ?*)						SEL(GVL.IOVD.Z_Man_Insu_Tst.e,
(*DEFAULT VALUE assignment*)							0,
(*ERROR is active*)										16#FE),
(*NOT AVAILABLE is active*)								16#FF),
(*Transmission is VALID*)								USINT_TO_BYTE(REAL_TO_USINT((GVL.IOVD.Z_Man_Insu_Tst.x))));
{endregion}

{region " SIGNAL AREA : NAME->Z_Semi_Aut_Insu_Tst LENGTH->8 STARTBIT :16"}
_FB_CanTx_Message_Unpack_485.X_Byte_2:=					SEL((GVL.IOVD.Z_Semi_Aut_Insu_Tst.v AND NOT GVL.IOVD.Z_Semi_Aut_Insu_Tst.RangeExcd),
(*SELECT 2 : Is NOT AVAILABLE ?*)						SEL(GVL.IOVD.Z_Semi_Aut_Insu_Tst.na,
(*SELECT 3 : Is ERROR active ?*)						SEL(GVL.IOVD.Z_Semi_Aut_Insu_Tst.e,
(*DEFAULT VALUE assignment*)							0,
(*ERROR is active*)										16#FE),
(*NOT AVAILABLE is active*)								16#FF),
(*Transmission is VALID*)								USINT_TO_BYTE(REAL_TO_USINT((GVL.IOVD.Z_Semi_Aut_Insu_Tst.x))));
{endregion}

{region " SIGNAL AREA : NAME->S_Insu_Tst_Ok LENGTH->1 STARTBIT :24"}
_FB_CanTx_Message_Unpack_485.S_Bit_24		:= GVL.IOVD.S_Insu_Tst_Ok.x AND GVL.IOVD.S_Insu_Tst_Ok.v;
{endregion}

{region " SIGNAL AREA : NAME->S_Man_Insu_Meas_Actv LENGTH->1 STARTBIT :25"}
_FB_CanTx_Message_Unpack_485.S_Bit_25		:= GVL.IOVD.S_Man_Insu_Meas_Actv.x AND GVL.IOVD.S_Man_Insu_Meas_Actv.v;
{endregion}

{region " SIGNAL AREA : NAME->S_Aut_Insu_Meas_Actv LENGTH->1 STARTBIT :26"}
_FB_CanTx_Message_Unpack_485.S_Bit_27		:= GVL.IOVD.S_Aut_Insu_Meas_Actv.x AND GVL.IOVD.S_Aut_Insu_Meas_Actv.v;
{endregion}

_FB_CanTx_Message_Unpack_485.S_Bit_5		:= TRUE;
_FB_CanTx_Message_Unpack_485.S_Bit_6		:= TRUE;
_FB_CanTx_Message_Unpack_485.S_Bit_7		:= TRUE;
_FB_CanTx_Message_Unpack_485.S_Bit_29		:= TRUE;
_FB_CanTx_Message_Unpack_485.S_Bit_30		:= TRUE;
_FB_CanTx_Message_Unpack_485.S_Bit_31		:= TRUE;
_FB_CanTx_Message_Unpack_485.X_Byte_4		:= 16#FF;
_FB_CanTx_Message_Unpack_485.X_Byte_5		:= 16#FF;
_FB_CanTx_Message_Unpack_485.X_Byte_6		:= 16#FF;
_FB_CanTx_Message_Unpack_485.X_Byte_7		:= 16#FF;

_FB_CanTx_Message_Unpack_485 (		C_Enable		:= GVL.IOVD.C_En_Isolation_Status_0X485,
     								Obj_CAN			:= ADR(GVL.IC.Obj_CAN0),
     								X_MsgID			:= 16#485,
     								Tm_CycleTime	:= TIME#250MS,
     								N_Msg_Dlc		:= 8,
     								S_Extended		:= 0,
     								S_Sent_Ok   	=> GVL.IOVD.S_SentOk_Isolation_Status_0X485);
{endregion}
//-----------------------------------------------------------------------------------------------------------------------------
//-----------------------------------------------------------------------------------------------------------------------------
{region " MESSAGE AREA :Arac_Genel_Istatistik- ID:4C2"}

{region " SIGNAL AREA : NAME->X_Spd_TCU LENGTH->8 STARTBIT :0"}
_FB_CanTx_Message_4C2.X_Byte_0							:=
(*SELECT 1 : Is data valid and range is not exceed?*)	SEL((GVL.IOVD.X_Spd_TCU.v AND NOT GVL.IOVD.X_Spd_TCU.RangeExcd),
(*SELECT 2 : Is NOT AVAILABLE ?*)						SEL(GVL.IOVD.X_Spd_TCU.na,
(*SELECT 3 : Is ERROR active ?*)						SEL(GVL.IOVD.X_Spd_TCU.e,
(*DEFAULT VALUE assignment*)							0,
(*ERROR is active*)										16#FE),
(*NOT AVAILABLE is active*)								16#FF),
(*Transmission is VALID*)								USINT_TO_BYTE(REAL_TO_USINT((GVL.IOVD.X_Spd_TCU.x))));
{endregion}

{region " SIGNAL AREA : NAME->X_Spd_EBS LENGTH->8 STARTBIT :8"}
_FB_CanTx_Message_4C2.X_Byte_1							:=
(*SELECT 1 : Is data valid and range is not exceed?*)	SEL((GVL.IOVD.X_Spd_EBS.v AND NOT GVL.IOVD.X_Spd_EBS.RangeExcd),
(*SELECT 2 : Is NOT AVAILABLE ?*)						SEL(GVL.IOVD.X_Spd_EBS.na,
(*SELECT 3 : Is ERROR active ?*)						SEL(GVL.IOVD.X_Spd_EBS.e,
(*DEFAULT VALUE assignment*)							0,
(*ERROR is active*)										16#FE),
(*NOT AVAILABLE is active*)								16#FF),
(*Transmission is VALID*)								USINT_TO_BYTE(REAL_TO_USINT((GVL.IOVD.X_Spd_EBS.x))));
{endregion}

{region " SIGNAL AREA : NAME->X_SOC LENGTH->8 STARTBIT :16"}
_FB_CanTx_Message_4C2.X_Byte_2							:=
(*SELECT 1 : Is data valid and range is not exceed?*)	SEL((GVL.IOVD.X_SOC.v AND NOT GVL.IOVD.X_SOC.RangeExcd),
(*SELECT 2 : Is NOT AVAILABLE ?*)						SEL(GVL.IOVD.X_SOC.na,
(*SELECT 3 : Is ERROR active ?*)						SEL(GVL.IOVD.X_SOC.e,
(*DEFAULT VALUE assignment*)							0,
(*ERROR is active*)										16#FE),
(*NOT AVAILABLE is active*)								16#FF),
(*Transmission is VALID*)								USINT_TO_BYTE(REAL_TO_USINT((GVL.IOVD.X_SOC.x))));
{endregion}

{region " SIGNAL AREA : NAME->X_SOH LENGTH->8 STARTBIT :24"}
_FB_CanTx_Message_4C2.X_Byte_3							:=
(*SELECT 1 : Is data valid and range is not exceed?*)	SEL((GVL.IOVD.X_SOH.v AND NOT GVL.IOVD.X_SOH.RangeExcd),
(*SELECT 2 : Is NOT AVAILABLE ?*)						SEL(GVL.IOVD.X_SOH.na,
(*SELECT 3 : Is ERROR active ?*)						SEL(GVL.IOVD.X_SOH.e,
(*DEFAULT VALUE assignment*)							0,
(*ERROR is active*)										16#FE),
(*NOT AVAILABLE is active*)								16#FF),
(*Transmission is VALID*)								USINT_TO_BYTE(REAL_TO_USINT((GVL.IOVD.X_SOH.x))));
{endregion}

{region " SIGNAL AREA : NAME->X_Accl LENGTH->16 STARTBIT :32"}
_FB_UNPACK_WORD_TO_BYTE_24 (	X_WORD_0	:= 
(*SELECT 1 : Is data valid and range is not exceed?*)	SEL((GVL.IOVD.X_Accl.v AND NOT GVL.IOVD.X_Accl.RangeExcd),
(*SELECT 2 : Is NOT AVAILABLE ?*)						SEL(GVL.IOVD.X_Accl.na,
(*SELECT 3 : Is ERROR active ?*)						SEL(GVL.IOVD.X_Accl.e,
(*DEFAULT VALUE assignment*)							UINT_TO_WORD(REAL_TO_UINT((32)/0.001)),
(*ERROR is active*)										16#FEFE),
(*NOT AVAILABLE is active*)								16#FFFF),
(*Transmission is VALID*)								UINT_TO_WORD(REAL_TO_UINT((GVL.IOVD.X_Accl.x + 32)/0.001))),
								X_BYTE_0	=> _FB_CanTx_Message_4C2.X_Byte_4,
								X_BYTE_1	=> _FB_CanTx_Message_4C2.X_Byte_5);
{endregion}

{region " SIGNAL AREA : NAME->X_Cosu_Avg LENGTH->16 STARTBIT :48"}
_FB_UNPACK_WORD_TO_BYTE_25 (
		X_WORD_0										:= 
(*SELECT 1 : Is data valid and range is not exceed?*)	SEL((GVL.IOVD.X_Cosu_Avg.v AND NOT GVL.IOVD.X_Cosu_Avg.RangeExcd),
(*SELECT 2 : Is NOT AVAILABLE ?*)						SEL(GVL.IOVD.X_Cosu_Avg.na,
(*SELECT 3 : Is ERROR active ?*)						SEL(GVL.IOVD.X_Cosu_Avg.e,
(*DEFAULT VALUE assignment*)							0,
(*ERROR is active*)										16#FEFE),
(*NOT AVAILABLE is active*)								16#FFFF),
(*Transmission is VALID*)								UINT_TO_WORD(REAL_TO_UINT((GVL.IOVD.X_Cosu_Avg.x)/0.001))),
		X_BYTE_0										=> _FB_CanTx_Message_4C2.X_Byte_6,
		X_BYTE_1										=> _FB_CanTx_Message_4C2.X_Byte_7);
{endregion}

_FB_CanTx_Message_4C2 (		C_Enable		:= GVL.IOVD.C_En_Arac_Genel_Istatistik_0X4C2,
     						Obj_CAN			:= ADR(GVL.IC.Obj_CAN0),
     						X_MsgID			:= 16#4C2,
     						Tm_CycleTime	:= TIME#250MS,
     						N_Msg_Dlc		:= 8,
     						S_Extended		:= 0,
     						S_Sent_Ok   	=> GVL.IOVD.S_SentOk_Arac_Genel_Istatistik_0X4C2);
{endregion}
//-----------------------------------------------------------------------------------------------------------------------------
//-----------------------------------------------------------------------------------------------------------------------------
{region " MESSAGE AREA :Temel_Durum- ID:99"}

{region " SIGNAL AREA : NAME->N_ECU_Lf LENGTH->8 STARTBIT :0"}
_FB_CanTx_Message_Unpack_99.X_Byte_0		:=
(*SELECT 1 : Is data valid and range is not exceed?*)	SEL((GVL.IOVD.N_ECU_Lf.v AND NOT GVL.IOVD.N_ECU_Lf.RangeExcd),
(*SELECT 2 : Is NOT AVAILABLE ?*)						SEL(GVL.IOVD.N_ECU_Lf.na,
(*SELECT 3 : Is ERROR active ?*)						SEL(GVL.IOVD.N_ECU_Lf.e,
(*DEFAULT VALUE assignment*)							0,
(*ERROR is active*)										16#FE),
(*NOT AVAILABLE is active*)								16#FF),
(*Transmission is VALID*)								USINT_TO_BYTE(GVL.IOVD.N_ECU_Lf.x ));

{endregion}

// PR1006_SRS_001391_TIMTRO
{region " SIGNAL AREA : NAME->S_Sw_Up_Avl LENGTH->2 STARTBIT :8"}
_FB_CanTx_Message_Unpack_99.S_Bit_8		:=	 (GVL.IOVD.S_Sw_Up_Avl.x OR GVL.IOVD.S_Sw_Up_Avl.na) AND NOT GVL.IOVD.S_Sw_Up_Avl.e; 
_FB_CanTx_Message_Unpack_99.S_Bit_9		:=	 NOT GVL.IOVD.S_Sw_Up_Avl.v OR GVL.IOVD.S_Sw_Up_Avl.na OR GVL.IOVD.S_Sw_Up_Avl.e; 

{endregion}

{region " SIGNAL AREA : NAME->S_EH_Rd_Avl LENGTH->2 STARTBIT :10"}
_FB_CanTx_Message_Unpack_99.S_Bit_10		:=	 (GVL.IOVD.S_EH_Rd_Avl.x OR GVL.IOVD.S_EH_Rd_Avl.na) AND NOT GVL.IOVD.S_EH_Rd_Avl.e; 
_FB_CanTx_Message_Unpack_99.S_Bit_11		:=	 NOT GVL.IOVD.S_EH_Rd_Avl.v OR GVL.IOVD.S_EH_Rd_Avl.na OR GVL.IOVD.S_EH_Rd_Avl.e; 

{endregion}

{region " SIGNAL AREA : NAME->S_Tst_Avl LENGTH->2 STARTBIT :12"}
_FB_CanTx_Message_Unpack_99.S_Bit_12		:=	 (GVL.IOVD.S_Tst_Avl.x OR GVL.IOVD.S_Tst_Avl.na) AND NOT GVL.IOVD.S_Tst_Avl.e; 
_FB_CanTx_Message_Unpack_99.S_Bit_13		:=	 NOT GVL.IOVD.S_Tst_Avl.v OR GVL.IOVD.S_Tst_Avl.na OR GVL.IOVD.S_Tst_Avl.e; 

{endregion}

{region " SIGNAL AREA : NAME->S_Para_Up_Avl LENGTH->2 STARTBIT :14"}
_FB_CanTx_Message_Unpack_99.S_Bit_14		:=	 (GVL.IOVD.S_Para_Up_Avl.x OR GVL.IOVD.S_Para_Up_Avl.na) AND NOT GVL.IOVD.S_Para_Up_Avl.e; 
_FB_CanTx_Message_Unpack_99.S_Bit_15		:=	 NOT GVL.IOVD.S_Para_Up_Avl.v OR GVL.IOVD.S_Para_Up_Avl.na OR GVL.IOVD.S_Para_Up_Avl.e; 

{endregion}

{region " SIGNAL AREA : NAME->C_ECU_Rst LENGTH->2 STARTBIT :16"}
_FB_CanTx_Message_Unpack_99.S_Bit_16		:=	 (GVL.IOVD.C_ECU_Rst.x OR GVL.IOVD.C_ECU_Rst.na) AND NOT GVL.IOVD.C_ECU_Rst.e; 
_FB_CanTx_Message_Unpack_99.S_Bit_17		:=	 NOT GVL.IOVD.C_ECU_Rst.v OR GVL.IOVD.C_ECU_Rst.na OR GVL.IOVD.C_ECU_Rst.e; 

{endregion}
{region " SIGNAL AREA : NAME->S_Brk_Tst_Mode LENGTH->2 STARTBIT :18"}
_FB_CanTx_Message_Unpack_99.S_Bit_18		:=	 (GVL.IOVD.S_Brk_Tst_Mode.x OR GVL.IOVD.S_Brk_Tst_Mode.na) AND NOT GVL.IOVD.S_Brk_Tst_Mode.e; 
_FB_CanTx_Message_Unpack_99.S_Bit_19		:=	 NOT GVL.IOVD.S_Brk_Tst_Mode.v OR GVL.IOVD.S_Brk_Tst_Mode.na OR GVL.IOVD.S_Brk_Tst_Mode.e; 

{endregion}
		  
{region " SIGNAL AREA : NAME->Z_Vh_Typ LENGTH->8 STARTBIT :32"}
_FB_CanTx_Message_Unpack_99.X_Byte_4		:=
(*SELECT 1 : Is data valid and range is not exceed?*)	SEL((GVL.IOVD.Z_Vh_Typ.v AND NOT GVL.IOVD.Z_Vh_Typ.RangeExcd),
(*SELECT 2 : Is NOT AVAILABLE ?*)						SEL(GVL.IOVD.Z_Vh_Typ.na,
(*SELECT 3 : Is ERROR active ?*)						SEL(GVL.IOVD.Z_Vh_Typ.e,
(*DEFAULT VALUE assignment*)							0,
(*ERROR is active*)										16#E),
(*NOT AVAILABLE is active*)								16#F),
(*Transmission is VALID*)								GVL.IOVD.Z_Vh_Typ.x);
{endregion}

// PR1006_SRS_001386_TIMTRO
{region " SIGNAL AREA : NAME->X_Prj_No LENGTH->16 STARTBIT->48}
_FB_UNPACK_WORD_TO_BYTE_30	(	X_Word_0				:=  
(*SELECT 1: Is data valid and range is not exceed?*)	SEL((GVL.IOVD.X_Prj_No.v AND NOT GVL.IOVD.X_Prj_No.RangeExcd),
(*SELECT 2: Is NOT AVAILABLE ?*)						SEL(GVL.IOVD.X_Prj_No.na,
(*SELECT 3: Is ERROR active ?*)							SEL(GVL.IOVD.X_Prj_No.e,
(*DEFAULT VALUE assignment*)							1000,
(*ERROR is active*)										16#FEFF),
(*NOT AVAILABLE is active*)								16#FFFF),
(*Transmission is VALID*)								UINT_TO_WORD(REAL_TO_UINT(GVL.IOVD.X_Prj_No.x))),
														X_Byte_0=> _FB_CanTx_Message_Unpack_99.X_Byte_6,
														X_Byte_1=> _FB_CanTx_Message_Unpack_99.X_Byte_7);
{endregion}
  
_FB_CanTx_Message_Unpack_99.S_Bit_22:=TRUE;
_FB_CanTx_Message_Unpack_99.S_Bit_23:=TRUE;
_FB_CanTx_Message_Unpack_99.X_Byte_3:=16#FF;
_FB_CanTx_Message_Unpack_99.X_Byte_5:=16#FF;
_FB_CanTx_Message_Unpack_99(
     C_Enable:= GVL.IOVD.C_En_Temel_Durum_0X99,
     Obj_CAN:= ADR(GVL.IC.Obj_CAN0),
     X_MsgID:= 16#99,
     Tm_CycleTime:= TIME#250ms,
     N_Msg_Dlc:=8,
     S_Extended:= 0,
     S_Sent_Ok   => GVL.IOVD.S_SentOk_Temel_Durum_0X99);
{endregion}
	 
	 
{region " MESSAGE AREA :Olay_Durum- ID:500"}

// PR1006_SRS_001881_TIMTRO
{region " SIGNAL AREA : NAME->X_Tot_TypA_Evnt LENGTH->16 STARTBIT :0"}
_FB_UNPACK_WORD_TO_BYTE_28(
		X_WORD_0:= 
(*SELECT 1 : Is data valid and range is not exceed?*)	SEL((GVL.IOVD.X_Tot_TypA_Evnt.v AND NOT GVL.IOVD.X_Tot_TypA_Evnt.RangeExcd),
(*SELECT 2 : Is NOT AVAILABLE ?*)						SEL(GVL.IOVD.X_Tot_TypA_Evnt.na,
(*SELECT 3 : Is ERROR active ?*)						SEL(GVL.IOVD.X_Tot_TypA_Evnt.e,
(*DEFAULT VALUE assignment*)							 0,
(*ERROR is active*)										16#FEFE),
(*NOT AVAILABLE is active*)								16#FFFF),
(*Transmission is VALID*)								UINT_TO_WORD(REAL_TO_UINT((GVL.IOVD.X_Tot_TypA_Evnt.x)))),
		X_BYTE_0=> _FB_CanTx_Message_500.X_Byte_0,
		X_BYTE_1=> _FB_CanTx_Message_500.X_Byte_1);
{endregion}

// PR1006_SRS_001881_TIMTRO
{region " SIGNAL AREA : NAME->X_Tot_TypB_Evnt LENGTH->16 STARTBIT :16"}
_FB_UNPACK_WORD_TO_BYTE_29(
		X_WORD_0:= 
(*SELECT 1 : Is data valid and range is not exceed?*)	SEL((GVL.IOVD.X_Tot_TypB_Evnt.v AND NOT GVL.IOVD.X_Tot_TypB_Evnt.RangeExcd),
(*SELECT 2 : Is NOT AVAILABLE ?*)						SEL(GVL.IOVD.X_Tot_TypB_Evnt.na,
(*SELECT 3 : Is ERROR active ?*)						SEL(GVL.IOVD.X_Tot_TypB_Evnt.e,
(*DEFAULT VALUE assignment*)							 0,
(*ERROR is active*)										16#FEFE),
(*NOT AVAILABLE is active*)								16#FFFF),
(*Transmission is VALID*)								UINT_TO_WORD(REAL_TO_UINT((GVL.IOVD.X_Tot_TypB_Evnt.x)))),
		X_BYTE_0=> _FB_CanTx_Message_500.X_Byte_2,
		X_BYTE_1=> _FB_CanTx_Message_500.X_Byte_3);
{endregion}
		  
_FB_CanTx_Message_500.X_Byte_4 := 16#FF;
_FB_CanTx_Message_500.X_Byte_5 := 16#FF;
_FB_CanTx_Message_500.X_Byte_6 := 16#FF;
_FB_CanTx_Message_500.X_Byte_7 := 16#FF;

_FB_CanTx_Message_500(	C_Enable := GVL.IOVD.C_En_Olay_Durum_0X500,
		 				Obj_CAN := ADR(GVL.IC.Obj_CAN0),
						X_MsgID := 16#500,
						Tm_CycleTime := T#250MS,
						N_Msg_Dlc := 8,
						S_Extended := FALSE,
						S_Sent_Ok => GVL.IOVD.S_SentOk_Olay_Durum_0X500);

{endregion}
//-----------------------------------------------------------------------------------------------------------------------------
                  
END_PROGRAM

PROGRAM P_IOVD_Set_Cycle

                    // 250ms cycle time
GVL.IOVD.C_En_Temel_Durum_0X99						:= GVL.SY.X_Cyc_Cnt = 1;
GVL.IOVD.C_En_ECU_Haberlesme_0X400 					:= GVL.IC.S_Diag_250ms_Actv AND GVL.SY.X_Cyc_Cnt = 1;
GVL.IOVD.C_En_DDS_0X401								:= GVL.IC.S_Diag_250ms_Actv AND GVL.SY.X_Cyc_Cnt = 1;
GVL.IOVD.C_En_DDS_2_0X402							:= GVL.IC.S_Diag_250ms_Actv AND GVL.SY.X_Cyc_Cnt = 1;
GVL.IOVD.C_En_HV_Durum_0X450						:= GVL.IC.S_Diag_250ms_Actv AND GVL.SY.X_Cyc_Cnt = 1;
GVL.IOVD.C_En_TCU_Ebus_Durum_0X461					:= GVL.IC.S_Diag_250ms_Actv AND GVL.SY.X_Cyc_Cnt = 1;
GVL.IOVD.C_En_TCU_Trolleybus_Durum_0X460			:= GVL.IC.S_Diag_250ms_Actv AND GVL.SY.X_Cyc_Cnt = 1;
GVL.IOVD.C_En_Olay_Durum_0X500						:= GVL.IC.S_Diag_250ms_Actv AND GVL.SY.X_Cyc_Cnt = 1;

GVL.IOVD.C_En_TCU_Surus_Limit_0X462					:= GVL.IC.S_Diag_250ms_Actv AND GVL.SY.X_Cyc_Cnt = 2;
GVL.IOVD.C_En_TCU_Analog_0X463						:= GVL.IC.S_Diag_250ms_Actv AND GVL.SY.X_Cyc_Cnt = 2;
GVL.IOVD.C_En_TCU_Cikis_Akim_Guc_0X464				:= GVL.IC.S_Diag_250ms_Actv AND GVL.SY.X_Cyc_Cnt = 2;
GVL.IOVD.C_En_TCU_Tork_Hiz_0X465					:= GVL.IC.S_Diag_250ms_Actv AND GVL.SY.X_Cyc_Cnt = 2;
GVL.IOVD.C_En_TCU_Calisma_Suresi_0X466				:= GVL.IC.S_Diag_250ms_Actv AND GVL.SY.X_Cyc_Cnt = 2;
GVL.IOVD.C_En_TCU_Analog_2_0X467					:= GVL.IC.S_Diag_250ms_Actv AND GVL.SY.X_Cyc_Cnt = 2;
GVL.IOVD.C_En_Yardimci_Konvertor_Durum_0X480		:= GVL.IC.S_Diag_250ms_Actv AND GVL.SY.X_Cyc_Cnt = 2;

GVL.IOVD.C_En_Yardimci_Konvertor_Akim_0X481			:= GVL.IC.S_Diag_250ms_Actv AND GVL.SY.X_Cyc_Cnt = 3;
GVL.IOVD.C_En_Yardimci_Konvertor_Guc_0X482			:= GVL.IC.S_Diag_250ms_Actv AND GVL.SY.X_Cyc_Cnt = 3;
GVL.IOVD.C_En_Batarya_Sarj_Konvertor_Analog_0X483	:= GVL.IC.S_Diag_250ms_Actv AND GVL.SY.X_Cyc_Cnt = 3;
GVL.IOVD.C_En_Yardimci_Konvertor_Sicaklik_0X484		:= GVL.IC.S_Diag_250ms_Actv AND GVL.SY.X_Cyc_Cnt = 3;
GVL.IOVD.C_En_Isolation_Status_0X485				:= GVL.IC.S_Diag_250ms_Actv AND GVL.SY.X_Cyc_Cnt = 3;
GVL.IOVD.C_En_Arac_Genel_Istatistik_0X4C2			:= GVL.IC.S_Diag_250ms_Actv AND GVL.SY.X_Cyc_Cnt = 3;

// 500ms cycle time
GVL.IOVD.C_En_ESS_Durum_0X430						:= GVL.IC.S_Diag_500ms_Actv AND GVL.SY.X_Cyc_Cnt_2 = 0;
GVL.IOVD.C_En_ESS_Paket_Voltaji_0X431				:= GVL.IC.S_Diag_500ms_Actv AND GVL.SY.X_Cyc_Cnt_2 = 0;
GVL.IOVD.C_En_ESS_Paket_Akim_0X432					:= GVL.IC.S_Diag_500ms_Actv AND GVL.SY.X_Cyc_Cnt_2 = 0;
GVL.IOVD.C_En_ESS_Maksimum_Hucre_Voltaji_0X433		:= GVL.IC.S_Diag_500ms_Actv AND GVL.SY.X_Cyc_Cnt_2 = 0;

GVL.IOVD.C_En_ESS_Minimum_Hucre_Voltaji_0X434		:= GVL.IC.S_Diag_500ms_Actv AND GVL.SY.X_Cyc_Cnt_2 = 1;
GVL.IOVD.C_En_ESS_Ortalama_Hucre_Voltaji_0X435		:= GVL.IC.S_Diag_500ms_Actv AND GVL.SY.X_Cyc_Cnt_2 = 1;
GVL.IOVD.C_En_ESS_Sicaklik_0X436					:= GVL.IC.S_Diag_500ms_Actv AND GVL.SY.X_Cyc_Cnt_2 = 1;
GVL.IOVD.C_En_ESS_Analog_0X437						:= GVL.IC.S_Diag_500ms_Actv AND GVL.SY.X_Cyc_Cnt_2 = 1;

GVL.IOVD.C_En_ESS_Sogutma_Suyu_0X438				:= GVL.IC.S_Diag_500ms_Actv AND GVL.SY.X_Cyc_Cnt_2 = 2;
GVL.IOVD.C_En_Sarj_Durum_0X4A0						:= GVL.IC.S_Diag_500ms_Actv AND GVL.SY.X_Cyc_Cnt_2 = 2;
GVL.IOVD.C_En_Sarj_Sureleri_0X4A5					:= GVL.IC.S_Diag_500ms_Actv AND GVL.SY.X_Cyc_Cnt_2 = 2;
GVL.IOVD.C_En_Sarj_Durum_3_0X4A6					:= GVL.IC.S_Diag_500ms_Actv AND GVL.SY.X_Cyc_Cnt_2 = 2;

GVL.IOVD.C_En_Pantograph_Analog_4_0X4AF				:= GVL.IC.S_Diag_500ms_Actv AND GVL.SY.X_Cyc_Cnt_2 = 3;
GVL.IOVD.C_En_Left_Charge_Analog_1_0X4B0			:= GVL.IC.S_Diag_500ms_Actv AND GVL.SY.X_Cyc_Cnt_2 = 3;
GVL.IOVD.C_En_Hava_Kompresoru_Durum_0X4F0			:= GVL.IC.S_Diag_500ms_Actv AND GVL.SY.X_Cyc_Cnt_2 = 3;

// 1000ms cycle time
GVL.IOVD.C_En_ECU_Parametre_0X403					:= GVL.IC.S_Diag_1000ms_Actv AND GVL.SY.X_Cyc_Cnt_1 = 0;
GVL.IOVD.C_En_HVAC_Durum_0X410						:= GVL.IC.S_Diag_1000ms_Actv AND GVL.SY.X_Cyc_Cnt_1 = 0;
GVL.IOVD.C_En_HVAC_Sicaklik_0X411					:= GVL.IC.S_Diag_1000ms_Actv AND GVL.SY.X_Cyc_Cnt_1 = 0;
GVL.IOVD.C_En_HVAC_Analog_0X413						:= GVL.IC.S_Diag_1000ms_Actv AND GVL.SY.X_Cyc_Cnt_1 = 0;
GVL.IOVD.C_En_Klima_Kontaktor_Kontrol_0X414			:= GVL.IC.S_Diag_1000ms_Actv AND GVL.SY.X_Cyc_Cnt_1 = 0;
GVL.IOVD.C_En_HVAC_Parameters_1_0X415				:= GVL.IC.S_Diag_1000ms_Actv AND GVL.SY.X_Cyc_Cnt_1 = 0;
GVL.IOVD.C_En_HVAC_Water_Temperature_0X416			:= GVL.IC.S_Diag_1000ms_Actv AND GVL.SY.X_Cyc_Cnt_1 = 0;

GVL.IOVD.C_En_Arac_Menzil_0X4C0						:= GVL.IC.S_Diag_1000ms_Actv AND GVL.SY.X_Cyc_Cnt_1 = 1;
GVL.IOVD.C_En_Arac_Odometre_0X4C1					:= GVL.IC.S_Diag_1000ms_Actv AND GVL.SY.X_Cyc_Cnt_1 = 1;
GVL.IOVD.C_En_Arac_Surus_Enerji_0X4C3				:= GVL.IC.S_Diag_1000ms_Actv AND GVL.SY.X_Cyc_Cnt_1 = 1;
GVL.IOVD.C_En_Arac_Tuketilen_Enerji_1_0X4C4			:= GVL.IC.S_Diag_1000ms_Actv AND GVL.SY.X_Cyc_Cnt_1 = 1;
GVL.IOVD.C_En_Arac_Tuketilen_Enerji_2_0X4C5			:= GVL.IC.S_Diag_1000ms_Actv AND GVL.SY.X_Cyc_Cnt_1 = 1;
GVL.IOVD.C_En_Arac_Kapasite_0X4C6					:= GVL.IC.S_Diag_1000ms_Actv AND GVL.SY.X_Cyc_Cnt_1 = 1;
GVL.IOVD.C_En_Arac_Sureler_0X4C7					:= GVL.IC.S_Diag_1000ms_Actv AND GVL.SY.X_Cyc_Cnt_1 = 1;

GVL.IOVD.C_En_Arac_Toplam_Tuketilen_Enerji_0X4C8	:= GVL.IC.S_Diag_1000ms_Actv AND GVL.SY.X_Cyc_Cnt_1 = 2;
GVL.IOVD.C_En_Arac_Genel_Istatistik_2_0X4C9			:= GVL.IC.S_Diag_1000ms_Actv AND GVL.SY.X_Cyc_Cnt_1 = 2;
GVL.IOVD.C_En_Klima_Calisma_Sureleri_1_0X4CA		:= GVL.IC.S_Diag_1000ms_Actv AND GVL.SY.X_Cyc_Cnt_1 = 2;
GVL.IOVD.C_En_Klima_Calisma_Sureleri_2_0X4CB		:= GVL.IC.S_Diag_1000ms_Actv AND GVL.SY.X_Cyc_Cnt_1 = 2;
GVL.IOVD.C_En_Sayicilar_1_0X4CC						:= GVL.IC.S_Diag_1000ms_Actv AND GVL.SY.X_Cyc_Cnt_1 = 2;
GVL.IOVD.C_En_Yardimci_Tuketici_Enerjileri_0X4CD	:= GVL.IC.S_Diag_1000ms_Actv AND GVL.SY.X_Cyc_Cnt_1 = 2;
GVL.IOVD.C_En_Kapi_Sayicilari_1_0X4CE				:= GVL.IC.S_Diag_1000ms_Actv AND GVL.SY.X_Cyc_Cnt_1 = 2;

GVL.IOVD.C_En_Kapi_Sayicilari_2_0X4CF				:= GVL.IC.S_Diag_1000ms_Actv AND GVL.SY.X_Cyc_Cnt_1 = 3;
GVL.IOVD.C_En_Sarj_Enerjisi_0X4D0					:= GVL.IC.S_Diag_1000ms_Actv AND GVL.SY.X_Cyc_Cnt_1 = 3;
GVL.IOVD.C_En_Arac_Bilgi_1_0X4E0					:= GVL.IC.S_Diag_1000ms_Actv AND GVL.SY.X_Cyc_Cnt_1 = 3;
GVL.IOVD.C_En_Arac_Bilgi_2_0X4E1					:= GVL.IC.S_Diag_1000ms_Actv AND GVL.SY.X_Cyc_Cnt_1 = 3;	


                  
END_PROGRAM

FUNCTION_BLOCK _FB_Tools_TmCalc
  VAR_INPUT
    S_Tm_Calc_En : BOOL;
    S_Frq_Actv : BOOL;
    C_Tm_Rst : BOOL;
    C_Eep_Rd : BOOL;
    X_Eep : REAL;
  END_VAR
  VAR_OUTPUT
    X_Tm_Tot_Min : REAL;
    X_Tm_Tot_Sec : REAL;
    S_Eep_Rd_Ok : BOOL := FALSE;
  END_VAR
  VAR
    R_Frq : R_TRIG;
    X_Mem_Cnt : USINT := 0;  (* USED FOR CLEARING THE VARIABLES AFTER EEPROM READING TRIGGER *)
  END_VAR

                    S_Eep_Rd_Ok		:= FALSE;

IF C_Eep_Rd THEN
	X_Tm_Tot_Min := 0;
	X_Tm_Tot_Sec := 0;

	X_Mem_Cnt	:= X_Mem_Cnt + 1;
END_IF

//Get these values from eeprom
//Reading eeprom process only performs once
IF X_Mem_Cnt = 1 THEN
	X_Tm_Tot_Min	:= X_Eep;
	
	S_Eep_Rd_Ok		:= TRUE;
	X_Mem_Cnt		:= 0;
END_IF

IF S_Tm_Calc_En THEN
	
	R_Frq(CLK := S_Frq_Actv);
	
	IF R_Frq.Q THEN
			
		IF X_Tm_Tot_Sec >= 59 AND X_Tm_Tot_Min <= 65000 THEN	
			X_Tm_Tot_Min 	:= X_Tm_Tot_Min + 1;
			X_Tm_Tot_Sec 	:= 0;
		END_IF
		X_Tm_Tot_Sec := X_Tm_Tot_Sec + 1;
	END_IF
	
END_IF

IF C_Tm_Rst THEN
	X_Tm_Tot_Min := 0;
	X_Tm_Tot_Sec := 0;
END_IF
                  
END_FUNCTION_BLOCK

CONFIGURATION HY_TTC_580
  RESOURCE Application ON PLC
    {attribute 'qualified_only'}
    VAR_GLOBAL  (* GVL *)
      IC : IC_T;  (* Struct object variable for Controller power management functions *)
      IIVD : IIVD_T;  (* DIAG *)
      IOVD : IOVD_T;  (* DIAG *)
      Param_Cst : ARRAY[1..18] OF REAL;  (* Constant Parameter Values *)
    END_VAR
    TASK Task_50ms_VD(INTERVAL := T#50ms, PRIORITY := 2);
    PROGRAM P_IIVD WITH Task_50ms_VD : P_IIVD;
    PROGRAM P_IOVD_Set_Cycle WITH Task_50ms_VD : P_IOVD_Set_Cycle;
    PROGRAM P_IOVD_Param WITH Task_50ms_VD : P_IOVD_Param;
    PROGRAM P_IOVD_A WITH Task_50ms_VD : P_IOVD_A;
    PROGRAM P_IOVD_B WITH Task_50ms_VD : P_IOVD_B;
    PROGRAM P_IOVD_C WITH Task_50ms_VD : P_IOVD_C;
  END_RESOURCE
END_CONFIGURATION

CONFIGURATION CANs
END_CONFIGURATION

CONFIGURATION CAN0
END_CONFIGURATION

CONFIGURATION CAN1
END_CONFIGURATION

CONFIGURATION CAN2
END_CONFIGURATION

CONFIGURATION CAN3
END_CONFIGURATION

CONFIGURATION CAN4
END_CONFIGURATION

CONFIGURATION CAN5
END_CONFIGURATION

CONFIGURATION CAN6
END_CONFIGURATION

CONFIGURATION System
END_CONFIGURATION

CONFIGURATION Analog_Inputs_2Mode_10V
END_CONFIGURATION

CONFIGURATION Pin 107
END_CONFIGURATION

CONFIGURATION DIN_S_K_Tst_Iso_Btn
END_CONFIGURATION

CONFIGURATION Pin 131
END_CONFIGURATION

CONFIGURATION <Empty>
END_CONFIGURATION

CONFIGURATION Pin 108
END_CONFIGURATION

CONFIGURATION DIN_S_Iso_Op_Mod_Man
END_CONFIGURATION

CONFIGURATION Pin 132
END_CONFIGURATION

CONFIGURATION <Empty>
END_CONFIGURATION

CONFIGURATION Pin 109
END_CONFIGURATION

CONFIGURATION <Empty>
END_CONFIGURATION

CONFIGURATION Pin 133
END_CONFIGURATION

CONFIGURATION <Empty>
END_CONFIGURATION

CONFIGURATION Pin 110
END_CONFIGURATION

CONFIGURATION <Empty>
END_CONFIGURATION

CONFIGURATION Pin 134
END_CONFIGURATION

CONFIGURATION <Empty>
END_CONFIGURATION

CONFIGURATION Analog_Inputs_2Mode_32V
END_CONFIGURATION

CONFIGURATION Pin 111
END_CONFIGURATION

CONFIGURATION <Empty>
END_CONFIGURATION

CONFIGURATION Pin 135
END_CONFIGURATION

CONFIGURATION <Empty>
END_CONFIGURATION

CONFIGURATION Pin 112
END_CONFIGURATION

CONFIGURATION <Empty>
END_CONFIGURATION

CONFIGURATION Pin 136
END_CONFIGURATION

CONFIGURATION <Empty>
END_CONFIGURATION

CONFIGURATION Pin 113
END_CONFIGURATION

CONFIGURATION <Empty>
END_CONFIGURATION

CONFIGURATION Pin 137
END_CONFIGURATION

CONFIGURATION <Empty>
END_CONFIGURATION

CONFIGURATION Pin 114
END_CONFIGURATION

CONFIGURATION <Empty>
END_CONFIGURATION

CONFIGURATION Pin 138
END_CONFIGURATION

CONFIGURATION <Empty>
END_CONFIGURATION

CONFIGURATION Analog_Inputs_3Mode
END_CONFIGURATION

CONFIGURATION Pin 103
END_CONFIGURATION

CONFIGURATION ADC_X_T_BTMS_Wtr_Snsr_In_Sd
END_CONFIGURATION

CONFIGURATION Pin 127
END_CONFIGURATION

CONFIGURATION <Empty>
END_CONFIGURATION

CONFIGURATION Pin 104
END_CONFIGURATION

CONFIGURATION ADC_X_T_BTMS_Wtr_Snsr_Out_Sd
END_CONFIGURATION

CONFIGURATION Pin 128
END_CONFIGURATION

CONFIGURATION DIN_S_ECU_Cvr_Op
END_CONFIGURATION

CONFIGURATION Pin 105
END_CONFIGURATION

CONFIGURATION ADC_X_T_BTMS_Wtr_Snr_In_Sd_Frnt_Md
END_CONFIGURATION

CONFIGURATION Pin 129
END_CONFIGURATION

CONFIGURATION DIN_S_MBMS_Cvr_Op
END_CONFIGURATION

CONFIGURATION Pin 106
END_CONFIGURATION

CONFIGURATION ADC_X_T_BTMS_Wtr_Snsr_Out_Sd_Frnt_Md
END_CONFIGURATION

CONFIGURATION Pin 130
END_CONFIGURATION

CONFIGURATION DIN_S_PDU_Cvr_Cl
END_CONFIGURATION

CONFIGURATION Digital_Outputs_HS
END_CONFIGURATION

CONFIGURATION Pin 149
END_CONFIGURATION

CONFIGURATION <Empty>
END_CONFIGURATION

CONFIGURATION Pin 173
END_CONFIGURATION

CONFIGURATION <Empty>
END_CONFIGURATION

CONFIGURATION Pin 152
END_CONFIGURATION

CONFIGURATION DIN_S_Em_Stop_Btn_Pres
END_CONFIGURATION

CONFIGURATION Pin 176
END_CONFIGURATION

CONFIGURATION DIN_S_B2_Actv
END_CONFIGURATION

CONFIGURATION Pin 155
END_CONFIGURATION

CONFIGURATION <Empty>
END_CONFIGURATION

CONFIGURATION Pin 179
END_CONFIGURATION

CONFIGURATION DIN_S_B4_Actv
END_CONFIGURATION

CONFIGURATION Pin 158
END_CONFIGURATION

CONFIGURATION DIN_S_B2_Actv_Fdbk
END_CONFIGURATION

CONFIGURATION Pin 182
END_CONFIGURATION

CONFIGURATION DIN_S_Em_Stop_Not_Actv_Fdbk
END_CONFIGURATION

CONFIGURATION Digital_Outputs_LS
END_CONFIGURATION

CONFIGURATION Pin 251
END_CONFIGURATION

CONFIGURATION <Empty>
END_CONFIGURATION

CONFIGURATION Pin 238
END_CONFIGURATION

CONFIGURATION <Empty>
END_CONFIGURATION

CONFIGURATION Pin 252
END_CONFIGURATION

CONFIGURATION <Empty>
END_CONFIGURATION

CONFIGURATION Pin 239
END_CONFIGURATION

CONFIGURATION <Empty>
END_CONFIGURATION

CONFIGURATION Pin 253
END_CONFIGURATION

CONFIGURATION <Empty>
END_CONFIGURATION

CONFIGURATION Pin 240
END_CONFIGURATION

CONFIGURATION DOUT_C_Tst_Iso_Led_Red
END_CONFIGURATION

CONFIGURATION Pin 254
END_CONFIGURATION

CONFIGURATION <Empty>
END_CONFIGURATION

CONFIGURATION Pin 241
END_CONFIGURATION

CONFIGURATION DOUT_C_K_Tst_Led_Grn
END_CONFIGURATION

CONFIGURATION PVG_Outputs
END_CONFIGURATION

CONFIGURATION Pin 161
END_CONFIGURATION

CONFIGURATION DOUT_C_Mot_Fan_Ct
END_CONFIGURATION

CONFIGURATION Pin 185
END_CONFIGURATION

CONFIGURATION <Empty>
END_CONFIGURATION

CONFIGURATION Pin 188
END_CONFIGURATION

CONFIGURATION <Empty>
END_CONFIGURATION

CONFIGURATION Pin 164
END_CONFIGURATION

CONFIGURATION <Empty>
END_CONFIGURATION

CONFIGURATION Pin 191
END_CONFIGURATION

CONFIGURATION <Empty>
END_CONFIGURATION

CONFIGURATION Pin 167
END_CONFIGURATION

CONFIGURATION DIN_S_Zero_Spd
END_CONFIGURATION

CONFIGURATION Pin 194
END_CONFIGURATION

CONFIGURATION <Empty>
END_CONFIGURATION

CONFIGURATION Pin 170
END_CONFIGURATION

CONFIGURATION DOUT_C_Air_Cmp_On
END_CONFIGURATION

CONFIGURATION PWM_Outputs
END_CONFIGURATION

CONFIGURATION Safety_switch_0
END_CONFIGURATION

CONFIGURATION Pin 153
END_CONFIGURATION

CONFIGURATION DOUT_C_BMS_Sp
END_CONFIGURATION

CONFIGURATION Pin 177
END_CONFIGURATION

CONFIGURATION <Empty>
END_CONFIGURATION

CONFIGURATION Pin 156
END_CONFIGURATION

CONFIGURATION <Empty>
END_CONFIGURATION

CONFIGURATION Pin 180
END_CONFIGURATION

CONFIGURATION <Empty>
END_CONFIGURATION

CONFIGURATION Pin 159
END_CONFIGURATION

CONFIGURATION <Empty>
END_CONFIGURATION

CONFIGURATION Pin 183
END_CONFIGURATION

CONFIGURATION <Empty>
END_CONFIGURATION

CONFIGURATION Pin 186
END_CONFIGURATION

CONFIGURATION <Empty>
END_CONFIGURATION

CONFIGURATION Pin 162
END_CONFIGURATION

CONFIGURATION <Empty>
END_CONFIGURATION

CONFIGURATION Pin 189
END_CONFIGURATION

CONFIGURATION DOUT_C_TCU_Sp
END_CONFIGURATION

CONFIGURATION Pin 165
END_CONFIGURATION

CONFIGURATION <Empty>
END_CONFIGURATION

CONFIGURATION Pin 192
END_CONFIGURATION

CONFIGURATION DIN_S_Prk_Brk
END_CONFIGURATION

CONFIGURATION Pin 168
END_CONFIGURATION

CONFIGURATION <Empty>
END_CONFIGURATION

CONFIGURATION Pin 195
END_CONFIGURATION

CONFIGURATION <Empty>
END_CONFIGURATION

CONFIGURATION Pin 171
END_CONFIGURATION

CONFIGURATION DOUT_C_TCU_STU_Sp
END_CONFIGURATION

CONFIGURATION Safety_switch_1
END_CONFIGURATION

CONFIGURATION Pin 154
END_CONFIGURATION

CONFIGURATION <Empty>
END_CONFIGURATION

CONFIGURATION Pin 178
END_CONFIGURATION

CONFIGURATION <Empty>
END_CONFIGURATION

CONFIGURATION Pin 157
END_CONFIGURATION

CONFIGURATION <Empty>
END_CONFIGURATION

CONFIGURATION Pin 181
END_CONFIGURATION

CONFIGURATION <Empty>
END_CONFIGURATION

CONFIGURATION Pin 160
END_CONFIGURATION

CONFIGURATION <Empty>
END_CONFIGURATION

CONFIGURATION Pin 184
END_CONFIGURATION

CONFIGURATION <Empty>
END_CONFIGURATION

CONFIGURATION Pin 187
END_CONFIGURATION

CONFIGURATION <Empty>
END_CONFIGURATION

CONFIGURATION Pin 163
END_CONFIGURATION

CONFIGURATION <Empty>
END_CONFIGURATION

CONFIGURATION Pin 190
END_CONFIGURATION

CONFIGURATION <Empty>
END_CONFIGURATION

CONFIGURATION Pin 166
END_CONFIGURATION

CONFIGURATION <Empty>
END_CONFIGURATION

CONFIGURATION Pin 193
END_CONFIGURATION

CONFIGURATION DIN_S_Mot_Fan_Fus_Blw
END_CONFIGURATION

CONFIGURATION Pin 169
END_CONFIGURATION

CONFIGURATION <Empty>
END_CONFIGURATION

CONFIGURATION Pin 196
END_CONFIGURATION

CONFIGURATION DIN_S_Air_Cmp_Thrm_Blw
END_CONFIGURATION

CONFIGURATION Pin 172
END_CONFIGURATION

CONFIGURATION <Empty>
END_CONFIGURATION

CONFIGURATION Safety_switch_2
END_CONFIGURATION

CONFIGURATION Pin 101
END_CONFIGURATION

CONFIGURATION DOUT_C_MBMS_Wkup
END_CONFIGURATION

CONFIGURATION Pin 125
END_CONFIGURATION

CONFIGURATION DOUT_C_TCU_Sft_Lp
END_CONFIGURATION

CONFIGURATION Pin 150
END_CONFIGURATION

CONFIGURATION <Empty>
END_CONFIGURATION

CONFIGURATION Pin 174
END_CONFIGURATION

CONFIGURATION <Empty>
END_CONFIGURATION

CONFIGURATION Pin 102
END_CONFIGURATION

CONFIGURATION DOUT_C_Heat_Sp
END_CONFIGURATION

CONFIGURATION Pin 126
END_CONFIGURATION

CONFIGURATION <Empty>
END_CONFIGURATION

CONFIGURATION Pin 151
END_CONFIGURATION

CONFIGURATION <Empty>
END_CONFIGURATION

CONFIGURATION Pin 175
END_CONFIGURATION

CONFIGURATION DOUT_C_MBMS_Sp
END_CONFIGURATION

CONFIGURATION Timer_Inputs_Cur
END_CONFIGURATION

CONFIGURATION Pin 115
END_CONFIGURATION

CONFIGURATION DIN_S_Mot_Fan_Deactv
END_CONFIGURATION

CONFIGURATION Pin 139
END_CONFIGURATION

CONFIGURATION <Empty>
END_CONFIGURATION

CONFIGURATION Pin 116
END_CONFIGURATION

CONFIGURATION DIN_S_Air_Cmp_Fus_Blw
END_CONFIGURATION

CONFIGURATION Pin 140
END_CONFIGURATION

CONFIGURATION DIN_S_AC_Chrg_Fus_Blw
END_CONFIGURATION

CONFIGURATION Pin 117
END_CONFIGURATION

CONFIGURATION DIN_S_Tacho_Spd_Pu_Out
END_CONFIGURATION

CONFIGURATION Pin 141
END_CONFIGURATION

CONFIGURATION DIN_S_AC_Fus_Blw
END_CONFIGURATION

CONFIGURATION Timer_Inputs
END_CONFIGURATION

CONFIGURATION Pin 122
END_CONFIGURATION

CONFIGURATION <Empty>
END_CONFIGURATION

CONFIGURATION Pin 146
END_CONFIGURATION

CONFIGURATION <Empty>
END_CONFIGURATION

CONFIGURATION Pin 123
END_CONFIGURATION

CONFIGURATION DIN_S_Air_Cmp_Ct_Deactv
END_CONFIGURATION

CONFIGURATION Pin 147
END_CONFIGURATION

CONFIGURATION <Empty>
END_CONFIGURATION

CONFIGURATION Pin 124
END_CONFIGURATION

CONFIGURATION DIN_S_Mot_Fan_Thrm_Ct
END_CONFIGURATION

CONFIGURATION Pin 148
END_CONFIGURATION

CONFIGURATION <Empty>
END_CONFIGURATION
